LIN {X 0,Y 525.54,Z 454.136,A -85,B 0,C 180,E1 -4756.393,E2 -4756.393} C_VEL
LIN {X 0,Y 525.32,Z 467.457,A -85,B 0,C 180,E1 -4756.732,E2 -4756.732} C_VEL
LIN {X 0,Y 525.04,Z 480.774,A -85,B 0,C 180,E1 -4757.241,E2 -4757.241} C_VEL
LIN {X 0,Y 524.811,Z 492.28,A -85,B 0,C 180,E1 -4757.845,E2 -4757.845} C_VEL
LIN {X 0,Y 524.533,Z 503.565,A -85,B 0,C 180,E1 -4758.602,E2 -4758.602} C_VEL
LIN {X 0,Y 524.201,Z 514.02,A -85,B 0,C 180,E1 -4759.475,E2 -4759.475} C_VEL
LIN {X 0,Y 523.995,Z 522.569,A -85,B 0,C 180,E1 -4760.349,E2 -4760.349} C_VEL
LIN {X 0,Y 523.801,Z 530.457,A -85,B 0,C 180,E1 -4761.319,E2 -4761.319} C_VEL
LIN {X 0,Y 523.605,Z 538.16,A -85,B 0,C 180,E1 -4762.481,E2 -4762.481} C_VEL
LIN {X 0,Y 523.482,Z 545.26,A -85,B 0,C 180,E1 -4763.835,E2 -4763.835} C_VEL
LIN {X 0,Y 523.383,Z 549.983,A -85,B 0,C 180,E1 -4764.993,E2 -4764.993} C_VEL
LIN {X 0,Y 523.443,Z 553.594,A -85,B 0,C 180,E1 -4766.151,E2 -4766.151} C_VEL
LIN {X 0,Y 523.367,Z 555.454,A -85,B 0,C 180,E1 -4766.922,E2 -4766.922} C_VEL
LIN {X 0,Y 523.334,Z 556.849,A -85,B 0,C 180,E1 -4767.692,E2 -4767.692} C_VEL
LIN {X 0,Y 523.25,Z 558.451,A -85,B 0,C 180,E1 -4769.231,E2 -4769.231} C_VEL
LIN {X 0,Y 523.247,Z 558.668,A -85,B 0,C 180,E1 -4770.001,E2 -4770.001} C_VEL
LIN {X 0,Y 523.274,Z 557.846,A -85,B 0,C 180,E1 -4771.54,E2 -4771.54} C_VEL
LIN {X 0,Y 523.334,Z 556.853,A -85,B 0,C 180,E1 -4772.31,E2 -4772.31} C_VEL
LIN {X 0,Y 523.368,Z 555.459,A -85,B 0,C 180,E1 -4773.08,E2 -4773.08} C_VEL
LIN {X 0,Y 523.424,Z 552.526,A -85,B 0,C 180,E1 -4774.236,E2 -4774.236} C_VEL
LIN {X 0,Y 523.462,Z 548.553,A -85,B 0,C 180,E1 -4775.393,E2 -4775.393} C_VEL
LIN {X 0,Y 523.513,Z 542.461,A -85,B 0,C 180,E1 -4776.743,E2 -4776.743} C_VEL
LIN {X 0,Y 523.667,Z 535.765,A -85,B 0,C 180,E1 -4777.907,E2 -4777.907} C_VEL
LIN {X 0,Y 523.88,Z 527.479,A -85,B 0,C 180,E1 -4779.07,E2 -4779.07} C_VEL
LIN {X 0,Y 524.073,Z 518.984,A -85,B 0,C 180,E1 -4780.041,E2 -4780.041} C_VEL
LIN {X 0,Y 524.352,Z 508.487,A -85,B 0,C 180,E1 -4781.012,E2 -4781.012} C_VEL
LIN {X 0,Y 524.635,Z 498.224,A -85,B 0,C 180,E1 -4781.78,E2 -4781.78} C_VEL
LIN {X 0,Y 524.943,Z 486.717,A -85,B 0,C 180,E1 -4782.468,E2 -4782.468} C_VEL
LIN {X 0,Y 525.177,Z 475.022,A -85,B 0,C 180,E1 -4783.003,E2 -4783.003} C_VEL
LIN {X 0,Y 525.4,Z 461.544,A -85,B 0,C 180,E1 -4783.44,E2 -4783.44} C_VEL
LIN {X 0,Y 525.581,Z 448.167,A -85,B 0,C 180,E1 -4783.706,E2 -4783.706} C_VEL
LIN {X 0,Y 525.774,Z 355.707,A -85,B 0,C 180,E1 -4784.979,E2 -4784.979} C_VEL
LIN {X 0,Y 524.311,Z 345.996,A -85,B 0,C 180,E1 -4785.179,E2 -4785.179} C_VEL
LIN {X 0,Y 524.7,Z 326.093,A -85,B 0,C 180,E1 -4788.307,E2 -4788.307} C_VEL
LIN {X 0,Y 525.163,Z 306.772,A -85,B 0,C 180,E1 -4791.388,E2 -4791.388} C_VEL
LIN {X 0,Y 525.315,Z 297.867,A -85,B 0,C 180,E1 -4792.829,E2 -4792.829} C_VEL
LIN {X 0,Y 523.939,Z 290.22,A -85,B 0,C 180,E1 -4794.171,E2 -4794.171} C_VEL
LIN {X 0,Y 523.949,Z 290.218,A -85,B 0,C 180,E1 -4797.134,E2 -4797.134} C_VEL
LIN {X 0,Y 523.94,Z 290.224,A -85,B 0,C 180,E1 -4799.757,E2 -4799.757} C_VEL
LIN {X 0,Y 523.937,Z 290.217,A -85,B 0,C 180,E1 -4802.45,E2 -4802.45} C_VEL
LIN {X 0,Y 523.921,Z 290.217,A -85,B 0,C 180,E1 -4805.227,E2 -4805.227} C_VEL
LIN {X 0,Y 523.917,Z 290.228,A -85,B 0,C 180,E1 -4808.102,E2 -4808.102} C_VEL
LIN {X 0,Y 523.943,Z 290.214,A -85,B 0,C 180,E1 -4811.308,E2 -4811.308} C_VEL
LIN {X 0,Y 523.942,Z 290.219,A -85,B 0,C 180,E1 -4814.689,E2 -4814.689} C_VEL
LIN {X 0,Y 523.947,Z 290.215,A -85,B 0,C 180,E1 -4817.88,E2 -4817.88} C_VEL
LIN {X 0,Y 523.922,Z 290.222,A -85,B 0,C 180,E1 -4820.915,E2 -4820.915} C_VEL
LIN {X 0,Y 523.899,Z 290.22,A -85,B 0,C 180,E1 -4823.825,E2 -4823.825} C_VEL
LIN {X 0,Y 523.945,Z 290.221,A -85,B 0,C 180,E1 -4826.636,E2 -4826.636} C_VEL
LIN {X 0,Y 523.952,Z 290.216,A -85,B 0,C 180,E1 -4829.355,E2 -4829.355} C_VEL
LIN {X 0,Y 523.95,Z 290.214,A -85,B 0,C 180,E1 -4832.288,E2 -4832.288} C_VEL
LIN {X 0,Y 523.906,Z 290.224,A -85,B 0,C 180,E1 -4835.427,E2 -4835.427} C_VEL
LIN {X 0,Y 523.941,Z 290.215,A -85,B 0,C 180,E1 -4837.939,E2 -4837.939} C_VEL
LIN {X 0,Y 523.977,Z 290.21,A -85,B 0,C 180,E1 -4840.408,E2 -4840.408} C_VEL
LIN {X 0,Y 523.958,Z 290.214,A -85,B 0,C 180,E1 -4842.837,E2 -4842.837} C_VEL
LIN {X 0,Y 523.98,Z 290.214,A -85,B 0,C 180,E1 -4845.236,E2 -4845.236} C_VEL
LIN {X 0,Y 524.017,Z 290.206,A -85,B 0,C 180,E1 -4848.394,E2 -4848.394} C_VEL
LIN {X 0,Y 523.964,Z 290.217,A -85,B 0,C 180,E1 -4851.515,E2 -4851.515} C_VEL
LIN {X 0,Y 524.036,Z 290.213,A -85,B 0,C 180,E1 -4853.841,E2 -4853.841} C_VEL
LIN {X 0,Y 524.035,Z 290.203,A -85,B 0,C 180,E1 -4856.925,E2 -4856.925} C_VEL
LIN {X 0,Y 524.118,Z 290.201,A -85,B 0,C 180,E1 -4860,E2 -4860} C_VEL
LIN {X 0,Y 524.04,Z 290.202,A -85,B 0,C 180,E1 -4863.075,E2 -4863.075} C_VEL
LIN {X 0,Y 524.013,Z 290.212,A -85,B 0,C 180,E1 -4866.159,E2 -4866.159} C_VEL
LIN {X 0,Y 523.989,Z 290.209,A -85,B 0,C 180,E1 -4869.262,E2 -4869.262} C_VEL
LIN {X 0,Y 524.003,Z 290.207,A -85,B 0,C 180,E1 -4871.737,E2 -4871.737} C_VEL
LIN {X 0,Y 523.997,Z 290.212,A -85,B 0,C 180,E1 -4875.052,E2 -4875.052} C_VEL
LIN {X 0,Y 523.95,Z 290.213,A -85,B 0,C 180,E1 -4877.969,E2 -4877.969} C_VEL
LIN {X 0,Y 523.975,Z 290.213,A -85,B 0,C 180,E1 -4880.41,E2 -4880.41} C_VEL
LIN {X 0,Y 523.912,Z 290.227,A -85,B 0,C 180,E1 -4882.893,E2 -4882.893} C_VEL
LIN {X 0,Y 523.931,Z 290.22,A -85,B 0,C 180,E1 -4885.42,E2 -4885.42} C_VEL
LIN {X 0,Y 523.92,Z 290.217,A -85,B 0,C 180,E1 -4888.002,E2 -4888.002} C_VEL
LIN {X 0,Y 523.941,Z 290.218,A -85,B 0,C 180,E1 -4890.853,E2 -4890.853} C_VEL
LIN {X 0,Y 523.932,Z 290.22,A -85,B 0,C 180,E1 -4893.729,E2 -4893.729} C_VEL
LIN {X 0,Y 523.901,Z 290.219,A -85,B 0,C 180,E1 -4896.4,E2 -4896.4} C_VEL
LIN {X 0,Y 523.922,Z 290.219,A -85,B 0,C 180,E1 -4899.084,E2 -4899.084} C_VEL
LIN {X 0,Y 523.942,Z 290.218,A -85,B 0,C 180,E1 -4902.12,E2 -4902.12} C_VEL
LIN {X 0,Y 523.945,Z 290.216,A -85,B 0,C 180,E1 -4905.31,E2 -4905.31} C_VEL
LIN {X 0,Y 523.902,Z 290.219,A -85,B 0,C 180,E1 -4906.901,E2 -4906.901} C_VEL
LIN {X 0,Y 523.239,Z 290.307,A -85,B 0,C 180,E1 -4907.542,E2 -4907.542} C_VEL
LIN {X 0,Y 520.398,Z 290.666,A -85,B 0,C 180,E1 -4908.584,E2 -4908.584} C_VEL
LIN {X 0,Y 517.994,Z 290.968,A -85,B 0,C 180,E1 -4909.423,E2 -4909.423} C_VEL
LIN {X 0,Y 516.958,Z 291.094,A -85,B 0,C 180,E1 -4910.071,E2 -4910.071} C_VEL
LIN {X 0,Y 516.872,Z 291.101,A -85,B 0,C 180,E1 -4910.29,E2 -4910.29} C_VEL
LIN {X 0,Y 516.854,Z 291.097,A -85,B 0,C 180,E1 -4913.346,E2 -4913.346} C_VEL
LIN {X 0,Y 516.908,Z 291.098,A -85,B 0,C 180,E1 -4916.12,E2 -4916.12} C_VEL
LIN {X 0,Y 516.893,Z 291.094,A -85,B 0,C 180,E1 -4918.935,E2 -4918.935} C_VEL
LIN {X 0,Y 516.865,Z 291.096,A -85,B 0,C 180,E1 -4921.581,E2 -4921.581} C_VEL
LIN {X 0,Y 516.881,Z 291.098,A -85,B 0,C 180,E1 -4924.208,E2 -4924.208} C_VEL
LIN {X 0,Y 516.858,Z 291.105,A -85,B 0,C 180,E1 -4926.775,E2 -4926.775} C_VEL
LIN {X 0,Y 516.939,Z 291.087,A -85,B 0,C 180,E1 -4929.732,E2 -4929.732} C_VEL
LIN {X 0,Y 516.896,Z 291.097,A -85,B 0,C 180,E1 -4932.594,E2 -4932.594} C_VEL
LIN {X 0,Y 516.941,Z 291.096,A -85,B 0,C 180,E1 -4935.029,E2 -4935.029} C_VEL
LIN {X 0,Y 516.967,Z 291.083,A -85,B 0,C 180,E1 -4938.233,E2 -4938.233} C_VEL
LIN {X 0,Y 516.952,Z 291.095,A -85,B 0,C 180,E1 -4941.399,E2 -4941.399} C_VEL
LIN {X 0,Y 516.994,Z 291.241,A -85,B 0,C 180,E1 -4943.471,E2 -4943.471} C_VEL
LIN {X 0,Y 517.644,Z 295.731,A -85,B 0,C 180,E1 -4944.35,E2 -4944.35} C_VEL
LIN {X 0,Y 517.356,Z 311.337,A -85,B 0,C 180,E1 -4947.274,E2 -4947.274} C_VEL
LIN {X 0,Y 517.208,Z 318.952,A -85,B 0,C 180,E1 -4948.685,E2 -4948.685} C_VEL
LIN {X 0,Y 519.149,Z 330.137,A -85,B 0,C 180,E1 -4948.908,E2 -4948.908} C_VEL
LIN {X 0,Y 518.644,Z 426.311,A -85,B 0,C 180,E1 -4950.266,E2 -4950.266} C_VEL
LIN {X 0,Y 518.412,Z 439.308,A -85,B 0,C 180,E1 -4950.606,E2 -4950.606} C_VEL
LIN {X 0,Y 518.173,Z 452.352,A -85,B 0,C 180,E1 -4951.116,E2 -4951.116} C_VEL
LIN {X 0,Y 517.881,Z 464.151,A -85,B 0,C 180,E1 -4951.749,E2 -4951.749} C_VEL
LIN {X 0,Y 517.553,Z 475.474,A -85,B 0,C 180,E1 -4952.529,E2 -4952.529} C_VEL
LIN {X 0,Y 517.309,Z 485.684,A -85,B 0,C 180,E1 -4953.407,E2 -4953.407} C_VEL
LIN {X 0,Y 517.029,Z 494.082,A -85,B 0,C 180,E1 -4954.287,E2 -4954.287} C_VEL
LIN {X 0,Y 516.728,Z 503.204,A -85,B 0,C 180,E1 -4955.462,E2 -4955.462} C_VEL
LIN {X 0,Y 516.566,Z 510.863,A -85,B 0,C 180,E1 -4956.695,E2 -4956.695} C_VEL
LIN {X 0,Y 516.442,Z 516.464,A -85,B 0,C 180,E1 -4957.821,E2 -4957.821} C_VEL
LIN {X 0,Y 516.333,Z 521.149,A -85,B 0,C 180,E1 -4959.005,E2 -4959.005} C_VEL
LIN {X 0,Y 516.303,Z 524.725,A -85,B 0,C 180,E1 -4960.192,E2 -4960.192} C_VEL
LIN {X 0,Y 516.263,Z 527.383,A -85,B 0,C 180,E1 -4961.435,E2 -4961.435} C_VEL
LIN {X 0,Y 516.177,Z 528.894,A -85,B 0,C 180,E1 -4962.582,E2 -4962.582} C_VEL
LIN {X 0,Y 516.175,Z 529.466,A -85,B 0,C 180,E1 -4963.382,E2 -4963.382} C_VEL
LIN {X 0,Y 516.247,Z 529.374,A -85,B 0,C 180,E1 -4964.858,E2 -4964.858} C_VEL
LIN {X 0,Y 516.159,Z 528.598,A -85,B 0,C 180,E1 -4965.801,E2 -4965.801} C_VEL
LIN {X 0,Y 516.187,Z 527.466,A -85,B 0,C 180,E1 -4966.613,E2 -4966.613} C_VEL
LIN {X 0,Y 516.267,Z 525.342,A -85,B 0,C 180,E1 -4967.652,E2 -4967.652} C_VEL
LIN {X 0,Y 516.346,Z 521.232,A -85,B 0,C 180,E1 -4969.066,E2 -4969.066} C_VEL
LIN {X 0,Y 516.45,Z 516.137,A -85,B 0,C 180,E1 -4970.344,E2 -4970.344} C_VEL
LIN {X 0,Y 516.573,Z 510.001,A -85,B 0,C 180,E1 -4971.551,E2 -4971.551} C_VEL
LIN {X 0,Y 516.82,Z 502.019,A -85,B 0,C 180,E1 -4972.802,E2 -4972.802} C_VEL
LIN {X 0,Y 517.058,Z 493.675,A -85,B 0,C 180,E1 -4973.851,E2 -4973.851} C_VEL
LIN {X 0,Y 517.304,Z 483.311,A -85,B 0,C 180,E1 -4974.907,E2 -4974.907} C_VEL
LIN {X 0,Y 517.621,Z 473.022,A -85,B 0,C 180,E1 -4975.751,E2 -4975.751} C_VEL
LIN {X 0,Y 517.986,Z 461.243,A -85,B 0,C 180,E1 -4976.513,E2 -4976.513} C_VEL
LIN {X 0,Y 518.215,Z 448.851,A -85,B 0,C 180,E1 -4977.13,E2 -4977.13} C_VEL
LIN {X 0,Y 518.466,Z 436.346,A -85,B 0,C 180,E1 -4977.58,E2 -4977.58} C_VEL
LIN {X 0,Y 518.663,Z 423.842,A -85,B 0,C 180,E1 -4977.87,E2 -4977.87} C_VEL
LIN {X 0,Y 518.99,Z 328.564,A -85,B 0,C 180,E1 -4979.209,E2 -4979.209} C_VEL
LIN {X 0,Y 517.258,Z 318.721,A -85,B 0,C 180,E1 -4979.422,E2 -4979.422} C_VEL
LIN {X 0,Y 517.456,Z 302.677,A -85,B 0,C 180,E1 -4982.31,E2 -4982.31} C_VEL
LIN {X 0,Y 517.383,Z 294.193,A -85,B 0,C 180,E1 -4983.843,E2 -4983.843} C_VEL
LIN {X 0,Y 516.905,Z 291.101,A -85,B 0,C 180,E1 -4984.445,E2 -4984.445} C_VEL
LIN {X 0,Y 516.855,Z 291.101,A -85,B 0,C 180,E1 -4987.725,E2 -4987.725} C_VEL
LIN {X 0,Y 516.857,Z 291.106,A -85,B 0,C 180,E1 -4990.743,E2 -4990.743} C_VEL
LIN {X 0,Y 516.847,Z 291.106,A -85,B 0,C 180,E1 -4992.834,E2 -4992.834} C_VEL
LIN {X 0,Y 516.888,Z 291.103,A -85,B 0,C 180,E1 -4995.006,E2 -4995.006} C_VEL
LIN {X 0,Y 516.879,Z 291.095,A -85,B 0,C 180,E1 -4998.402,E2 -4998.402} C_VEL
LIN {X 0,Y 516.868,Z 291.106,A -85,B 0,C 180,E1 -5001.283,E2 -5001.283} C_VEL
LIN {X 0,Y 516.862,Z 291.098,A -85,B 0,C 180,E1 -5004.219,E2 -5004.219} C_VEL
LIN {X 0,Y 516.872,Z 291.093,A -85,B 0,C 180,E1 -5007.052,E2 -5007.052} C_VEL
LIN {X 0,Y 516.873,Z 291.1,A -85,B 0,C 180,E1 -5009.795,E2 -5009.795} C_VEL
LIN {X 0,Y 516.866,Z 291.097,A -85,B 0,C 180,E1 -5012.464,E2 -5012.464} C_VEL
LIN {X 0,Y 516.862,Z 291.105,A -85,B 0,C 180,E1 -5015.645,E2 -5015.645} C_VEL
LIN {X 0,Y 516.875,Z 291.096,A -85,B 0,C 180,E1 -5018.462,E2 -5018.462} C_VEL
LIN {X 0,Y 516.878,Z 291.094,A -85,B 0,C 180,E1 -5020.954,E2 -5020.954} C_VEL
LIN {X 0,Y 516.824,Z 291.102,A -85,B 0,C 180,E1 -5023.407,E2 -5023.407} C_VEL
LIN {X 0,Y 516.861,Z 291.104,A -85,B 0,C 180,E1 -5025.833,E2 -5025.833} C_VEL
LIN {X 0,Y 516.915,Z 291.097,A -85,B 0,C 180,E1 -5028.233,E2 -5028.233} C_VEL
LIN {X 0,Y 516.907,Z 291.088,A -85,B 0,C 180,E1 -5031.399,E2 -5031.399} C_VEL
LIN {X 0,Y 516.964,Z 291.089,A -85,B 0,C 180,E1 -5034.539,E2 -5034.539} C_VEL
LIN {X 0,Y 517.054,Z 291.071,A -85,B 0,C 180,E1 -5037.663,E2 -5037.663} C_VEL
LIN {X 0,Y 517.078,Z 291.072,A -85,B 0,C 180,E1 -5040.779,E2 -5040.779} C_VEL
LIN {X 0,Y 516.931,Z 291.089,A -85,B 0,C 180,E1 -5043.118,E2 -5043.118} C_VEL
LIN {X 0,Y 516.97,Z 291.087,A -85,B 0,C 180,E1 -5046.244,E2 -5046.244} C_VEL
LIN {X 0,Y 516.909,Z 291.094,A -85,B 0,C 180,E1 -5048.602,E2 -5048.602} C_VEL
LIN {X 0,Y 516.943,Z 291.085,A -85,B 0,C 180,E1 -5051.807,E2 -5051.807} C_VEL
LIN {X 0,Y 516.926,Z 291.094,A -85,B 0,C 180,E1 -5055.143,E2 -5055.143} C_VEL
LIN {X 0,Y 516.903,Z 291.088,A -85,B 0,C 180,E1 -5058.223,E2 -5058.223} C_VEL
LIN {X 0,Y 516.896,Z 291.096,A -85,B 0,C 180,E1 -5060.702,E2 -5060.702} C_VEL
LIN {X 0,Y 516.876,Z 291.094,A -85,B 0,C 180,E1 -5064.074,E2 -5064.074} C_VEL
LIN {X 0,Y 516.838,Z 291.101,A -85,B 0,C 180,E1 -5066.663,E2 -5066.663} C_VEL
LIN {X 0,Y 516.899,Z 291.099,A -85,B 0,C 180,E1 -5069.523,E2 -5069.523} C_VEL
LIN {X 0,Y 516.889,Z 291.093,A -85,B 0,C 180,E1 -5072.544,E2 -5072.544} C_VEL
LIN {X 0,Y 516.857,Z 291.104,A -85,B 0,C 180,E1 -5075.33,E2 -5075.33} C_VEL
LIN {X 0,Y 516.871,Z 291.099,A -85,B 0,C 180,E1 -5077.943,E2 -5077.943} C_VEL
LIN {X 0,Y 516.859,Z 291.098,A -85,B 0,C 180,E1 -5080.744,E2 -5080.744} C_VEL
LIN {X 0,Y 516.853,Z 291.094,A -85,B 0,C 180,E1 -5082.835,E2 -5082.835} C_VEL
LIN {X 0,Y 516.89,Z 291.093,A -85,B 0,C 180,E1 -5085.008,E2 -5085.008} C_VEL
LIN {X 0,Y 516.905,Z 291.096,A -85,B 0,C 180,E1 -5088.4,E2 -5088.4} C_VEL
LIN {X 0,Y 516.875,Z 291.098,A -85,B 0,C 180,E1 -5091.285,E2 -5091.285} C_VEL
LIN {X 0,Y 516.864,Z 291.104,A -85,B 0,C 180,E1 -5094.22,E2 -5094.22} C_VEL
LIN {X 0,Y 516.892,Z 291.095,A -85,B 0,C 180,E1 -5097.054,E2 -5097.054} C_VEL
LIN {X 0,Y 516.884,Z 291.1,A -85,B 0,C 180,E1 -5099.797,E2 -5099.797} C_VEL
LIN {X 0,Y 516.92,Z 291.099,A -85,B 0,C 180,E1 -5102.468,E2 -5102.468} C_VEL
LIN {X 0,Y 516.926,Z 291.265,A -85,B 0,C 180,E1 -5105.779,E2 -5105.779} C_VEL
LIN {X 0,Y 518.335,Z 299.595,A -85,B 0,C 180,E1 -5107.221,E2 -5107.221} C_VEL
LIN {X 0,Y 517.928,Z 316.612,A -85,B 0,C 180,E1 -5109.977,E2 -5109.977} C_VEL
LIN {X 0,Y 517.489,Z 334.423,A -85,B 0,C 180,E1 -5112.82,E2 -5112.82} C_VEL
LIN {X 0,Y 517.275,Z 346.087,A -85,B 0,C 180,E1 -5114.637,E2 -5114.637} C_VEL
LIN {X 0,Y 519.095,Z 358.575,A -85,B 0,C 180,E1 -5114.867,E2 -5114.867} C_VEL
LIN {X 0,Y 518.636,Z 453.891,A -85,B 0,C 180,E1 -5116.208,E2 -5116.208} C_VEL
LIN {X 0,Y 518.422,Z 467.226,A -85,B 0,C 180,E1 -5116.552,E2 -5116.552} C_VEL
LIN {X 0,Y 518.131,Z 479.424,A -85,B 0,C 180,E1 -5117.018,E2 -5117.018} C_VEL
LIN {X 0,Y 517.867,Z 491.836,A -85,B 0,C 180,E1 -5117.665,E2 -5117.665} C_VEL
LIN {X 0,Y 517.552,Z 503.35,A -85,B 0,C 180,E1 -5118.447,E2 -5118.447} C_VEL
LIN {X 0,Y 517.203,Z 513.807,A -85,B 0,C 180,E1 -5119.331,E2 -5119.331} C_VEL
LIN {X 0,Y 516.962,Z 522.359,A -85,B 0,C 180,E1 -5120.217,E2 -5120.217} C_VEL
LIN {X 0,Y 516.729,Z 530.248,A -85,B 0,C 180,E1 -5121.199,E2 -5121.199} C_VEL
LIN {X 0,Y 516.544,Z 537.954,A -85,B 0,C 180,E1 -5122.378,E2 -5122.378} C_VEL
LIN {X 0,Y 516.418,Z 543.657,A -85,B 0,C 180,E1 -5123.449,E2 -5123.449} C_VEL
LIN {X 0,Y 516.375,Z 548.349,A -85,B 0,C 180,E1 -5124.534,E2 -5124.534} C_VEL
LIN {X 0,Y 516.312,Z 552.321,A -85,B 0,C 180,E1 -5125.707,E2 -5125.707} C_VEL
LIN {X 0,Y 516.282,Z 555.254,A -85,B 0,C 180,E1 -5126.879,E2 -5126.879} C_VEL
LIN {X 0,Y 516.26,Z 556.65,A -85,B 0,C 180,E1 -5127.66,E2 -5127.66} C_VEL
LIN {X 0,Y 516.16,Z 558.252,A -85,B 0,C 180,E1 -5129.221,E2 -5129.221} C_VEL
LIN {X 0,Y 516.155,Z 558.469,A -85,B 0,C 180,E1 -5130.001,E2 -5130.001} C_VEL
LIN {X 0,Y 516.192,Z 557.648,A -85,B 0,C 180,E1 -5131.561,E2 -5131.561} C_VEL
LIN {X 0,Y 516.26,Z 556.656,A -85,B 0,C 180,E1 -5132.341,E2 -5132.341} C_VEL
LIN {X 0,Y 516.283,Z 555.261,A -85,B 0,C 180,E1 -5133.122,E2 -5133.122} C_VEL
LIN {X 0,Y 516.312,Z 552.327,A -85,B 0,C 180,E1 -5134.294,E2 -5134.294} C_VEL
LIN {X 0,Y 516.376,Z 548.354,A -85,B 0,C 180,E1 -5135.468,E2 -5135.468} C_VEL
LIN {X 0,Y 516.422,Z 543.143,A -85,B 0,C 180,E1 -5136.664,E2 -5136.664} C_VEL
LIN {X 0,Y 516.582,Z 536.801,A -85,B 0,C 180,E1 -5137.82,E2 -5137.82} C_VEL
LIN {X 0,Y 516.786,Z 528.768,A -85,B 0,C 180,E1 -5138.998,E2 -5138.998} C_VEL
LIN {X 0,Y 517.018,Z 520.582,A -85,B 0,C 180,E1 -5139.981,E2 -5139.981} C_VEL
LIN {X 0,Y 517.326,Z 510.6,A -85,B 0,C 180,E1 -5140.965,E2 -5140.965} C_VEL
LIN {X 0,Y 517.629,Z 500.75,A -85,B 0,C 180,E1 -5141.752,E2 -5141.752} C_VEL
LIN {X 0,Y 517.917,Z 489.613,A -85,B 0,C 180,E1 -5142.465,E2 -5142.465} C_VEL
LIN {X 0,Y 518.178,Z 477.16,A -85,B 0,C 180,E1 -5143.082,E2 -5143.082} C_VEL
LIN {X 0,Y 518.439,Z 464.063,A -85,B 0,C 180,E1 -5143.549,E2 -5143.549} C_VEL
LIN {X 0,Y 518.659,Z 450.968,A -85,B 0,C 180,E1 -5143.843,E2 -5143.843} C_VEL
LIN {X 0,Y 518.991,Z 356.872,A -85,B 0,C 180,E1 -5145.16,E2 -5145.16} C_VEL
LIN {X 0,Y 517.289,Z 345.951,A -85,B 0,C 180,E1 -5145.366,E2 -5145.366} C_VEL
LIN {X 0,Y 517.746,Z 325.651,A -85,B 0,C 180,E1 -5148.603,E2 -5148.603} C_VEL
LIN {X 0,Y 518.203,Z 307.858,A -85,B 0,C 180,E1 -5151.481,E2 -5151.481} C_VEL
LIN {X 0,Y 518.355,Z 299.1,A -85,B 0,C 180,E1 -5152.915,E2 -5152.915} C_VEL
LIN {X 0,Y 516.884,Z 291.099,A -85,B 0,C 180,E1 -5154.317,E2 -5154.317} C_VEL
LIN {X 0,Y 516.926,Z 291.098,A -85,B 0,C 180,E1 -5157.533,E2 -5157.533} C_VEL
LIN {X 0,Y 516.89,Z 291.097,A -85,B 0,C 180,E1 -5160.204,E2 -5160.204} C_VEL
LIN {X 0,Y 516.899,Z 291.092,A -85,B 0,C 180,E1 -5162.947,E2 -5162.947} C_VEL
LIN {X 0,Y 516.871,Z 291.101,A -85,B 0,C 180,E1 -5165.781,E2 -5165.781} C_VEL
LIN {X 0,Y 516.881,Z 291.096,A -85,B 0,C 180,E1 -5168.716,E2 -5168.716} C_VEL
LIN {X 0,Y 516.905,Z 291.094,A -85,B 0,C 180,E1 -5171.776,E2 -5171.776} C_VEL
LIN {X 0,Y 516.899,Z 291.093,A -85,B 0,C 180,E1 -5175.007,E2 -5175.007} C_VEL
LIN {X 0,Y 516.914,Z 291.098,A -85,B 0,C 180,E1 -5178.399,E2 -5178.399} C_VEL
LIN {X 0,Y 516.882,Z 291.095,A -85,B 0,C 180,E1 -5181.284,E2 -5181.284} C_VEL
LIN {X 0,Y 516.871,Z 291.097,A -85,B 0,C 180,E1 -5184.219,E2 -5184.219} C_VEL
LIN {X 0,Y 516.899,Z 291.098,A -85,B 0,C 180,E1 -5187.053,E2 -5187.053} C_VEL
LIN {X 0,Y 516.89,Z 291.093,A -85,B 0,C 180,E1 -5189.796,E2 -5189.796} C_VEL
LIN {X 0,Y 516.903,Z 291.093,A -85,B 0,C 180,E1 -5192.466,E2 -5192.466} C_VEL
LIN {X 0,Y 516.849,Z 291.107,A -85,B 0,C 180,E1 -5195.068,E2 -5195.068} C_VEL
LIN {X 0,Y 516.873,Z 291.099,A -85,B 0,C 180,E1 -5197.621,E2 -5197.621} C_VEL
LIN {X 0,Y 516.935,Z 291.088,A -85,B 0,C 180,E1 -5200.13,E2 -5200.13} C_VEL
LIN {X 0,Y 516.909,Z 291.09,A -85,B 0,C 180,E1 -5202.595,E2 -5202.595} C_VEL
LIN {X 0,Y 516.946,Z 291.088,A -85,B 0,C 180,E1 -5205.03,E2 -5205.03} C_VEL
LIN {X 0,Y 516.97,Z 291.085,A -85,B 0,C 180,E1 -5208.234,E2 -5208.234} C_VEL
LIN {X 0,Y 516.939,Z 291.091,A -85,B 0,C 180,E1 -5211.399,E2 -5211.399} C_VEL
LIN {X 0,Y 517.002,Z 291.087,A -85,B 0,C 180,E1 -5213.757,E2 -5213.757} C_VEL
LIN {X 0,Y 517.084,Z 291.073,A -85,B 0,C 180,E1 -5217.663,E2 -5217.663} C_VEL
LIN {X 0,Y 517.091,Z 291.069,A -85,B 0,C 180,E1 -5220.779,E2 -5220.779} C_VEL
LIN {X 0,Y 516.983,Z 291.081,A -85,B 0,C 180,E1 -5223.117,E2 -5223.117} C_VEL
LIN {X 0,Y 516.978,Z 291.09,A -85,B 0,C 180,E1 -5226.243,E2 -5226.243} C_VEL
LIN {X 0,Y 516.944,Z 291.086,A -85,B 0,C 180,E1 -5229.389,E2 -5229.389} C_VEL
LIN {X 0,Y 516.955,Z 291.085,A -85,B 0,C 180,E1 -5231.807,E2 -5231.807} C_VEL
LIN {X 0,Y 516.95,Z 291.088,A -85,B 0,C 180,E1 -5235.147,E2 -5235.147} C_VEL
LIN {X 0,Y 516.918,Z 291.091,A -85,B 0,C 180,E1 -5238.222,E2 -5238.222} C_VEL
LIN {X 0,Y 516.915,Z 291.096,A -85,B 0,C 180,E1 -5240.701,E2 -5240.701} C_VEL
LIN {X 0,Y 516.891,Z 291.092,A -85,B 0,C 180,E1 -5244.073,E2 -5244.073} C_VEL
LIN {X 0,Y 516.9,Z 291.094,A -85,B 0,C 180,E1 -5246.659,E2 -5246.659} C_VEL
LIN {X 0,Y 516.911,Z 291.096,A -85,B 0,C 180,E1 -5249.523,E2 -5249.523} C_VEL
LIN {X 0,Y 516.896,Z 291.092,A -85,B 0,C 180,E1 -5252.543,E2 -5252.543} C_VEL
LIN {X 0,Y 516.866,Z 291.104,A -85,B 0,C 180,E1 -5255.329,E2 -5255.329} C_VEL
LIN {X 0,Y 516.881,Z 291.098,A -85,B 0,C 180,E1 -5257.942,E2 -5257.942} C_VEL
LIN {X 0,Y 516.882,Z 291.094,A -85,B 0,C 180,E1 -5260.742,E2 -5260.742} C_VEL
LIN {X 0,Y 516.883,Z 291.102,A -85,B 0,C 180,E1 -5263.903,E2 -5263.903} C_VEL
LIN {X 0,Y 516.85,Z 291.098,A -85,B 0,C 180,E1 -5266.902,E2 -5266.902} C_VEL
LIN {X 0,Y 516.886,Z 291.097,A -85,B 0,C 180,E1 -5269.589,E2 -5269.589} C_VEL
LIN {X 0,Y 516.872,Z 291.101,A -85,B 0,C 180,E1 -5270.29,E2 -5270.29} C_VEL
LIN {X 0,Y 516.201,Z 291.181,A -85,B 0,C 180,E1 -5270.94,E2 -5270.94} C_VEL
LIN {X 0,Y 513.347,Z 291.542,A -85,B 0,C 180,E1 -5271.996,E2 -5271.996} C_VEL
LIN {X 0,Y 510.934,Z 291.841,A -85,B 0,C 180,E1 -5272.846,E2 -5272.846} C_VEL
LIN {X 0,Y 509.894,Z 291.967,A -85,B 0,C 180,E1 -5273.503,E2 -5273.503} C_VEL
LIN {X 0,Y 509.807,Z 291.977,A -85,B 0,C 180,E1 -5273.725,E2 -5273.725} C_VEL
LIN {X 0,Y 509.86,Z 291.974,A -85,B 0,C 180,E1 -5276.539,E2 -5276.539} C_VEL
LIN {X 0,Y 509.847,Z 291.97,A -85,B 0,C 180,E1 -5279.334,E2 -5279.334} C_VEL
LIN {X 0,Y 509.852,Z 291.973,A -85,B 0,C 180,E1 -5282.051,E2 -5282.051} C_VEL
LIN {X 0,Y 509.809,Z 291.983,A -85,B 0,C 180,E1 -5284.7,E2 -5284.7} C_VEL
LIN {X 0,Y 509.826,Z 291.973,A -85,B 0,C 180,E1 -5287.458,E2 -5287.458} C_VEL
LIN {X 0,Y 509.916,Z 291.961,A -85,B 0,C 180,E1 -5289.844,E2 -5289.844} C_VEL
LIN {X 0,Y 509.865,Z 291.974,A -85,B 0,C 180,E1 -5293.173,E2 -5293.173} C_VEL
LIN {X 0,Y 509.857,Z 291.97,A -85,B 0,C 180,E1 -5295.633,E2 -5295.633} C_VEL
LIN {X 0,Y 509.909,Z 291.968,A -85,B 0,C 180,E1 -5298.874,E2 -5298.874} C_VEL
LIN {X 0,Y 509.92,Z 291.966,A -85,B 0,C 180,E1 -5302.077,E2 -5302.077} C_VEL
LIN {X 0,Y 509.958,Z 292.135,A -85,B 0,C 180,E1 -5303.343,E2 -5303.343} C_VEL
LIN {X 0,Y 510.664,Z 296.834,A -85,B 0,C 180,E1 -5304.273,E2 -5304.273} C_VEL
LIN {X 0,Y 510.379,Z 311.463,A -85,B 0,C 180,E1 -5307.039,E2 -5307.039} C_VEL
LIN {X 0,Y 510.242,Z 319.101,A -85,B 0,C 180,E1 -5308.47,E2 -5308.47} C_VEL
LIN {X 0,Y 512.269,Z 330.125,A -85,B 0,C 180,E1 -5308.697,E2 -5308.697} C_VEL
LIN {X 0,Y 511.753,Z 426.291,A -85,B 0,C 180,E1 -5310.073,E2 -5310.073} C_VEL
LIN {X 0,Y 511.534,Z 439.338,A -85,B 0,C 180,E1 -5310.417,E2 -5310.417} C_VEL
LIN {X 0,Y 511.263,Z 452.439,A -85,B 0,C 180,E1 -5310.935,E2 -5310.935} C_VEL
LIN {X 0,Y 510.938,Z 464.274,A -85,B 0,C 180,E1 -5311.576,E2 -5311.576} C_VEL
LIN {X 0,Y 510.584,Z 475.614,A -85,B 0,C 180,E1 -5312.366,E2 -5312.366} C_VEL
LIN {X 0,Y 510.319,Z 485.833,A -85,B 0,C 180,E1 -5313.256,E2 -5313.256} C_VEL
LIN {X 0,Y 510.003,Z 494.244,A -85,B 0,C 180,E1 -5314.148,E2 -5314.148} C_VEL
LIN {X 0,Y 509.749,Z 502.011,A -85,B 0,C 180,E1 -5315.141,E2 -5315.141} C_VEL
LIN {X 0,Y 509.577,Z 509.605,A -85,B 0,C 180,E1 -5316.334,E2 -5316.334} C_VEL
LIN {X 0,Y 509.41,Z 515.734,A -85,B 0,C 180,E1 -5317.53,E2 -5317.53} C_VEL
LIN {X 0,Y 509.278,Z 520.613,A -85,B 0,C 180,E1 -5318.73,E2 -5318.73} C_VEL
LIN {X 0,Y 509.23,Z 524.372,A -85,B 0,C 180,E1 -5319.933,E2 -5319.933} C_VEL
LIN {X 0,Y 509.174,Z 527.725,A -85,B 0,C 180,E1 -5321.48,E2 -5321.48} C_VEL
LIN {X 0,Y 509.099,Z 529.286,A -85,B 0,C 180,E1 -5322.76,E2 -5322.76} C_VEL
LIN {X 0,Y 509.085,Z 529.718,A -85,B 0,C 180,E1 -5323.572,E2 -5323.572} C_VEL
LIN {X 0,Y 509.148,Z 529.536,A -85,B 0,C 180,E1 -5324.93,E2 -5324.93} C_VEL
LIN {X 0,Y 509.063,Z 528.566,A -85,B 0,C 180,E1 -5326.028,E2 -5326.028} C_VEL
LIN {X 0,Y 509.105,Z 527.296,A -85,B 0,C 180,E1 -5326.851,E2 -5326.851} C_VEL
LIN {X 0,Y 509.197,Z 525.411,A -85,B 0,C 180,E1 -5327.76,E2 -5327.76} C_VEL
LIN {X 0,Y 509.264,Z 522.13,A -85,B 0,C 180,E1 -5328.923,E2 -5328.923} C_VEL
LIN {X 0,Y 509.393,Z 517.147,A -85,B 0,C 180,E1 -5330.252,E2 -5330.252} C_VEL
LIN {X 0,Y 509.484,Z 511.396,A -85,B 0,C 180,E1 -5331.44,E2 -5331.44} C_VEL
LIN {X 0,Y 509.738,Z 503.68,A -85,B 0,C 180,E1 -5332.708,E2 -5332.708} C_VEL
LIN {X 0,Y 509.978,Z 495.696,A -85,B 0,C 180,E1 -5333.771,E2 -5333.771} C_VEL
LIN {X 0,Y 510.298,Z 486.306,A -85,B 0,C 180,E1 -5334.793,E2 -5334.793} C_VEL
LIN {X 0,Y 510.617,Z 476.044,A -85,B 0,C 180,E1 -5335.693,E2 -5335.693} C_VEL
LIN {X 0,Y 510.936,Z 465.895,A -85,B 0,C 180,E1 -5336.413,E2 -5336.413} C_VEL
LIN {X 0,Y 511.232,Z 453.865,A -85,B 0,C 180,E1 -5337.088,E2 -5337.088} C_VEL
LIN {X 0,Y 511.447,Z 442.37,A -85,B 0,C 180,E1 -5337.574,E2 -5337.574} C_VEL
LIN {X 0,Y 511.682,Z 429.048,A -85,B 0,C 180,E1 -5337.959,E2 -5337.959} C_VEL
LIN {X 0,Y 511.847,Z 410.339,A -85,B 0,C 180,E1 -5338.262,E2 -5338.262} C_VEL
LIN {X 0,Y 512.232,Z 329.911,A -85,B 0,C 180,E1 -5339.398,E2 -5339.398} C_VEL
LIN {X 0,Y 510.249,Z 318.946,A -85,B 0,C 180,E1 -5339.624,E2 -5339.624} C_VEL
LIN {X 0,Y 510.471,Z 302.1,A -85,B 0,C 180,E1 -5342.68,E2 -5342.68} C_VEL
LIN {X 0,Y 510.413,Z 295.471,A -85,B 0,C 180,E1 -5343.893,E2 -5343.893} C_VEL
LIN {X 0,Y 509.861,Z 291.978,A -85,B 0,C 180,E1 -5344.591,E2 -5344.591} C_VEL
LIN {X 0,Y 509.81,Z 291.981,A -85,B 0,C 180,E1 -5347.34,E2 -5347.34} C_VEL
LIN {X 0,Y 509.811,Z 291.979,A -85,B 0,C 180,E1 -5350.384,E2 -5350.384} C_VEL
LIN {X 0,Y 509.794,Z 291.987,A -85,B 0,C 180,E1 -5353.059,E2 -5353.059} C_VEL
LIN {X 0,Y 509.814,Z 291.977,A -85,B 0,C 180,E1 -5355.793,E2 -5355.793} C_VEL
LIN {X 0,Y 509.823,Z 291.975,A -85,B 0,C 180,E1 -5358.571,E2 -5358.571} C_VEL
LIN {X 0,Y 509.841,Z 291.974,A -85,B 0,C 180,E1 -5361.786,E2 -5361.786} C_VEL
LIN {X 0,Y 509.82,Z 291.975,A -85,B 0,C 180,E1 -5364.621,E2 -5364.621} C_VEL
LIN {X 0,Y 509.851,Z 291.975,A -85,B 0,C 180,E1 -5367.48,E2 -5367.48} C_VEL
LIN {X 0,Y 509.849,Z 291.97,A -85,B 0,C 180,E1 -5370.274,E2 -5370.274} C_VEL
LIN {X 0,Y 509.811,Z 291.977,A -85,B 0,C 180,E1 -5372.94,E2 -5372.94} C_VEL
LIN {X 0,Y 509.824,Z 291.98,A -85,B 0,C 180,E1 -5375.572,E2 -5375.572} C_VEL
LIN {X 0,Y 509.812,Z 291.978,A -85,B 0,C 180,E1 -5378.148,E2 -5378.148} C_VEL
LIN {X 0,Y 509.844,Z 291.971,A -85,B 0,C 180,E1 -5380.681,E2 -5380.681} C_VEL
LIN {X 0,Y 509.778,Z 291.978,A -85,B 0,C 180,E1 -5383.171,E2 -5383.171} C_VEL
LIN {X 0,Y 509.834,Z 291.976,A -85,B 0,C 180,E1 -5385.633,E2 -5385.633} C_VEL
LIN {X 0,Y 509.879,Z 291.975,A -85,B 0,C 180,E1 -5388.131,E2 -5388.131} C_VEL
LIN {X 0,Y 509.861,Z 291.965,A -85,B 0,C 180,E1 -5391.279,E2 -5391.279} C_VEL
LIN {X 0,Y 509.884,Z 291.967,A -85,B 0,C 180,E1 -5393.669,E2 -5393.669} C_VEL
LIN {X 0,Y 509.873,Z 291.967,A -85,B 0,C 180,E1 -5396.84,E2 -5396.84} C_VEL
LIN {X 0,Y 509.916,Z 291.97,A -85,B 0,C 180,E1 -5398.421,E2 -5398.421} C_VEL
LIN {X 0,Y 510.027,Z 291.95,A -85,B 0,C 180,E1 -5400.79,E2 -5400.79} C_VEL
LIN {X 0,Y 509.875,Z 291.967,A -85,B 0,C 180,E1 -5403.161,E2 -5403.161} C_VEL
LIN {X 0,Y 509.924,Z 291.966,A -85,B 0,C 180,E1 -5406.33,E2 -5406.33} C_VEL
LIN {X 0,Y 509.842,Z 291.971,A -85,B 0,C 180,E1 -5409.522,E2 -5409.522} C_VEL
LIN {X 0,Y 509.895,Z 291.963,A -85,B 0,C 180,E1 -5411.932,E2 -5411.932} C_VEL
LIN {X 0,Y 509.886,Z 291.969,A -85,B 0,C 180,E1 -5415.242,E2 -5415.242} C_VEL
LIN {X 0,Y 509.847,Z 291.968,A -85,B 0,C 180,E1 -5418.484,E2 -5418.484} C_VEL
LIN {X 0,Y 509.837,Z 291.98,A -85,B 0,C 180,E1 -5421.002,E2 -5421.002} C_VEL
LIN {X 0,Y 509.81,Z 291.978,A -85,B 0,C 180,E1 -5423.565,E2 -5423.565} C_VEL
LIN {X 0,Y 509.811,Z 291.975,A -85,B 0,C 180,E1 -5426.358,E2 -5426.358} C_VEL
LIN {X 0,Y 509.842,Z 291.973,A -85,B 0,C 180,E1 -5428.847,E2 -5428.847} C_VEL
LIN {X 0,Y 509.811,Z 291.981,A -85,B 0,C 180,E1 -5431.591,E2 -5431.591} C_VEL
LIN {X 0,Y 509.84,Z 291.972,A -85,B 0,C 180,E1 -5434.415,E2 -5434.415} C_VEL
LIN {X 0,Y 509.801,Z 291.983,A -85,B 0,C 180,E1 -5437.342,E2 -5437.342} C_VEL
LIN {X 0,Y 509.812,Z 291.977,A -85,B 0,C 180,E1 -5440.385,E2 -5440.385} C_VEL
LIN {X 0,Y 509.799,Z 291.974,A -85,B 0,C 180,E1 -5443.061,E2 -5443.061} C_VEL
LIN {X 0,Y 509.818,Z 291.984,A -85,B 0,C 180,E1 -5445.794,E2 -5445.794} C_VEL
LIN {X 0,Y 509.848,Z 291.974,A -85,B 0,C 180,E1 -5448.575,E2 -5448.575} C_VEL
LIN {X 0,Y 509.846,Z 291.979,A -85,B 0,C 180,E1 -5451.788,E2 -5451.788} C_VEL
LIN {X 0,Y 509.824,Z 291.975,A -85,B 0,C 180,E1 -5454.623,E2 -5454.623} C_VEL
LIN {X 0,Y 509.859,Z 291.972,A -85,B 0,C 180,E1 -5457.482,E2 -5457.482} C_VEL
LIN {X 0,Y 509.856,Z 291.977,A -85,B 0,C 180,E1 -5460.275,E2 -5460.275} C_VEL
LIN {X 0,Y 509.872,Z 291.974,A -85,B 0,C 180,E1 -5462.945,E2 -5462.945} C_VEL
LIN {X 0,Y 509.853,Z 292.012,A -85,B 0,C 180,E1 -5465.574,E2 -5465.574} C_VEL
LIN {X 0,Y 511.359,Z 300.354,A -85,B 0,C 180,E1 -5467.049,E2 -5467.049} C_VEL
LIN {X 0,Y 511.014,Z 315.639,A -85,B 0,C 180,E1 -5469.569,E2 -5469.569} C_VEL
LIN {X 0,Y 510.503,Z 334.207,A -85,B 0,C 180,E1 -5472.578,E2 -5472.578} C_VEL
LIN {X 0,Y 510.239,Z 345.662,A -85,B 0,C 180,E1 -5474.416,E2 -5474.416} C_VEL
LIN {X 0,Y 512.255,Z 359.615,A -85,B 0,C 180,E1 -5474.678,E2 -5474.678} C_VEL
LIN {X 0,Y 511.761,Z 453.644,A -85,B 0,C 180,E1 -5476.019,E2 -5476.019} C_VEL
LIN {X 0,Y 511.523,Z 466.993,A -85,B 0,C 180,E1 -5476.367,E2 -5476.367} C_VEL
LIN {X 0,Y 511.174,Z 480.325,A -85,B 0,C 180,E1 -5476.889,E2 -5476.889} C_VEL
LIN {X 0,Y 510.903,Z 491.791,A -85,B 0,C 180,E1 -5477.506,E2 -5477.506} C_VEL
LIN {X 0,Y 510.57,Z 503.134,A -85,B 0,C 180,E1 -5478.286,E2 -5478.286} C_VEL
LIN {X 0,Y 510.212,Z 513.595,A -85,B 0,C 180,E1 -5479.183,E2 -5479.183} C_VEL
LIN {X 0,Y 509.94,Z 522.148,A -85,B 0,C 180,E1 -5480.081,E2 -5480.081} C_VEL
LIN {X 0,Y 509.681,Z 530.04,A -85,B 0,C 180,E1 -5481.077,E2 -5481.077} C_VEL
LIN {X 0,Y 509.479,Z 537.748,A -85,B 0,C 180,E1 -5482.271,E2 -5482.271} C_VEL
LIN {X 0,Y 509.318,Z 543.986,A -85,B 0,C 180,E1 -5483.474,E2 -5483.474} C_VEL
LIN {X 0,Y 509.243,Z 549.579,A -85,B 0,C 180,E1 -5484.854,E2 -5484.854} C_VEL
LIN {X 0,Y 509.245,Z 553.191,A -85,B 0,C 180,E1 -5486.044,E2 -5486.044} C_VEL
LIN {X 0,Y 509.2,Z 555.054,A -85,B 0,C 180,E1 -5486.836,E2 -5486.836} C_VEL
LIN {X 0,Y 509.189,Z 556.45,A -85,B 0,C 180,E1 -5487.628,E2 -5487.628} C_VEL
LIN {X 0,Y 509.073,Z 558.054,A -85,B 0,C 180,E1 -5489.21,E2 -5489.21} C_VEL
LIN {X 0,Y 509.066,Z 558.271,A -85,B 0,C 180,E1 -5490.001,E2 -5490.001} C_VEL
LIN {X 0,Y 509.112,Z 557.45,A -85,B 0,C 180,E1 -5491.583,E2 -5491.583} C_VEL
LIN {X 0,Y 509.189,Z 556.458,A -85,B 0,C 180,E1 -5492.374,E2 -5492.374} C_VEL
LIN {X 0,Y 509.201,Z 555.063,A -85,B 0,C 180,E1 -5493.165,E2 -5493.165} C_VEL
LIN {X 0,Y 509.204,Z 552.128,A -85,B 0,C 180,E1 -5494.354,E2 -5494.354} C_VEL
LIN {X 0,Y 509.293,Z 548.155,A -85,B 0,C 180,E1 -5495.544,E2 -5495.544} C_VEL
LIN {X 0,Y 509.397,Z 542.144,A -85,B 0,C 180,E1 -5496.914,E2 -5496.914} C_VEL
LIN {X 0,Y 509.545,Z 535.362,A -85,B 0,C 180,E1 -5498.128,E2 -5498.128} C_VEL
LIN {X 0,Y 509.783,Z 527.074,A -85,B 0,C 180,E1 -5499.323,E2 -5499.323} C_VEL
LIN {X 0,Y 510.016,Z 518.575,A -85,B 0,C 180,E1 -5500.32,E2 -5500.32} C_VEL
LIN {X 0,Y 510.395,Z 508.075,A -85,B 0,C 180,E1 -5501.317,E2 -5501.317} C_VEL
LIN {X 0,Y 510.688,Z 497.802,A -85,B 0,C 180,E1 -5502.107,E2 -5502.107} C_VEL
LIN {X 0,Y 511.05,Z 486.294,A -85,B 0,C 180,E1 -5502.813,E2 -5502.813} C_VEL
LIN {X 0,Y 511.359,Z 474.585,A -85,B 0,C 180,E1 -5503.361,E2 -5503.361} C_VEL
LIN {X 0,Y 511.592,Z 461.09,A -85,B 0,C 180,E1 -5503.81,E2 -5503.81} C_VEL
LIN {X 0,Y 511.819,Z 447.66,A -85,B 0,C 180,E1 -5504.082,E2 -5504.082} C_VEL
LIN {X 0,Y 512.17,Z 357.903,A -85,B 0,C 180,E1 -5505.35,E2 -5505.35} C_VEL
LIN {X 0,Y 510.259,Z 345.664,A -85,B 0,C 180,E1 -5505.597,E2 -5505.597} C_VEL
LIN {X 0,Y 510.755,Z 326.736,A -85,B 0,C 180,E1 -5508.659,E2 -5508.659} C_VEL
LIN {X 0,Y 511.252,Z 308.917,A -85,B 0,C 180,E1 -5511.576,E2 -5511.576} C_VEL
LIN {X 0,Y 511.433,Z 300.494,A -85,B 0,C 180,E1 -5512.971,E2 -5512.971} C_VEL
LIN {X 0,Y 509.856,Z 291.975,A -85,B 0,C 180,E1 -5514.473,E2 -5514.473} C_VEL
LIN {X 0,Y 509.878,Z 291.971,A -85,B 0,C 180,E1 -5517.057,E2 -5517.057} C_VEL
LIN {X 0,Y 509.861,Z 291.978,A -85,B 0,C 180,E1 -5519.751,E2 -5519.751} C_VEL
LIN {X 0,Y 509.877,Z 291.966,A -85,B 0,C 180,E1 -5522.774,E2 -5522.774} C_VEL
LIN {X 0,Y 509.826,Z 291.976,A -85,B 0,C 180,E1 -5525.578,E2 -5525.578} C_VEL
LIN {X 0,Y 509.852,Z 291.976,A -85,B 0,C 180,E1 -5528.338,E2 -5528.338} C_VEL
LIN {X 0,Y 509.848,Z 291.97,A -85,B 0,C 180,E1 -5531.427,E2 -5531.427} C_VEL
LIN {X 0,Y 509.843,Z 291.976,A -85,B 0,C 180,E1 -5534.67,E2 -5534.67} C_VEL
LIN {X 0,Y 509.854,Z 291.973,A -85,B 0,C 180,E1 -5538.104,E2 -5538.104} C_VEL
LIN {X 0,Y 509.849,Z 291.979,A -85,B 0,C 180,E1 -5540.647,E2 -5540.647} C_VEL
LIN {X 0,Y 509.813,Z 291.974,A -85,B 0,C 180,E1 -5543.646,E2 -5543.646} C_VEL
LIN {X 0,Y 509.862,Z 291.973,A -85,B 0,C 180,E1 -5546.539,E2 -5546.539} C_VEL
LIN {X 0,Y 509.846,Z 291.974,A -85,B 0,C 180,E1 -5549.334,E2 -5549.334} C_VEL
LIN {X 0,Y 509.854,Z 291.969,A -85,B 0,C 180,E1 -5552.052,E2 -5552.052} C_VEL
LIN {X 0,Y 509.807,Z 291.978,A -85,B 0,C 180,E1 -5554.7,E2 -5554.7} C_VEL
LIN {X 0,Y 509.829,Z 291.979,A -85,B 0,C 180,E1 -5557.458,E2 -5557.458} C_VEL
LIN {X 0,Y 509.92,Z 291.963,A -85,B 0,C 180,E1 -5559.845,E2 -5559.845} C_VEL
LIN {X 0,Y 509.876,Z 291.972,A -85,B 0,C 180,E1 -5563.174,E2 -5563.174} C_VEL
LIN {X 0,Y 509.864,Z 291.977,A -85,B 0,C 180,E1 -5565.634,E2 -5565.634} C_VEL
LIN {X 0,Y 509.915,Z 291.962,A -85,B 0,C 180,E1 -5568.874,E2 -5568.874} C_VEL
LIN {X 0,Y 509.918,Z 291.967,A -85,B 0,C 180,E1 -5572.078,E2 -5572.078} C_VEL
LIN {X 0,Y 509.977,Z 291.956,A -85,B 0,C 180,E1 -5574.464,E2 -5574.464} C_VEL
LIN {X 0,Y 510.053,Z 291.948,A -85,B 0,C 180,E1 -5577.631,E2 -5577.631} C_VEL
LIN {X 0,Y 510.06,Z 291.952,A -85,B 0,C 180,E1 -5580,E2 -5580} C_VEL
LIN {X 0,Y 510.052,Z 291.952,A -85,B 0,C 180,E1 -5582.369,E2 -5582.369} C_VEL
LIN {X 0,Y 509.966,Z 291.956,A -85,B 0,C 180,E1 -5585.536,E2 -5585.536} C_VEL
LIN {X 0,Y 509.912,Z 291.967,A -85,B 0,C 180,E1 -5588.72,E2 -5588.72} C_VEL
LIN {X 0,Y 509.908,Z 291.964,A -85,B 0,C 180,E1 -5591.931,E2 -5591.931} C_VEL
LIN {X 0,Y 509.897,Z 291.966,A -85,B 0,C 180,E1 -5595.242,E2 -5595.242} C_VEL
LIN {X 0,Y 509.863,Z 291.973,A -85,B 0,C 180,E1 -5598.483,E2 -5598.483} C_VEL
LIN {X 0,Y 509.853,Z 291.978,A -85,B 0,C 180,E1 -5601.001,E2 -5601.001} C_VEL
LIN {X 0,Y 509.823,Z 291.975,A -85,B 0,C 180,E1 -5603.564,E2 -5603.564} C_VEL
LIN {X 0,Y 509.882,Z 291.966,A -85,B 0,C 180,E1 -5606.371,E2 -5606.371} C_VEL
LIN {X 0,Y 509.86,Z 291.971,A -85,B 0,C 180,E1 -5609.726,E2 -5609.726} C_VEL
LIN {X 0,Y 509.869,Z 291.969,A -85,B 0,C 180,E1 -5612.773,E2 -5612.773} C_VEL
LIN {X 0,Y 509.825,Z 291.981,A -85,B 0,C 180,E1 -5615.578,E2 -5615.578} C_VEL
LIN {X 0,Y 509.851,Z 291.97,A -85,B 0,C 180,E1 -5618.338,E2 -5618.338} C_VEL
LIN {X 0,Y 509.853,Z 291.975,A -85,B 0,C 180,E1 -5621.426,E2 -5621.426} C_VEL
LIN {X 0,Y 509.841,Z 291.971,A -85,B 0,C 180,E1 -5624.67,E2 -5624.67} C_VEL
LIN {X 0,Y 509.852,Z 291.977,A -85,B 0,C 180,E1 -5628.104,E2 -5628.104} C_VEL
LIN {X 0,Y 509.839,Z 291.973,A -85,B 0,C 180,E1 -5630.646,E2 -5630.646} C_VEL
LIN {X 0,Y 509.807,Z 291.977,A -85,B 0,C 180,E1 -5633.725,E2 -5633.725} C_VEL
LIN {X 0,Y 509.148,Z 292.064,A -85,B 0,C 180,E1 -5634.385,E2 -5634.385} C_VEL
LIN {X 0,Y 506.343,Z 292.409,A -85,B 0,C 180,E1 -5635.457,E2 -5635.457} C_VEL
LIN {X 0,Y 503.957,Z 292.713,A -85,B 0,C 180,E1 -5636.321,E2 -5636.321} C_VEL
LIN {X 0,Y 502.909,Z 292.836,A -85,B 0,C 180,E1 -5636.987,E2 -5636.987} C_VEL
LIN {X 0,Y 502.811,Z 292.847,A -85,B 0,C 180,E1 -5637.213,E2 -5637.213} C_VEL
LIN {X 0,Y 502.817,Z 292.85,A -85,B 0,C 180,E1 -5640.065,E2 -5640.065} C_VEL
LIN {X 0,Y 502.845,Z 292.842,A -85,B 0,C 180,E1 -5643.443,E2 -5643.443} C_VEL
LIN {X 0,Y 502.788,Z 292.855,A -85,B 0,C 180,E1 -5646.959,E2 -5646.959} C_VEL
LIN {X 0,Y 502.835,Z 292.844,A -85,B 0,C 180,E1 -5649.548,E2 -5649.548} C_VEL
LIN {X 0,Y 502.818,Z 292.846,A -85,B 0,C 180,E1 -5652.091,E2 -5652.091} C_VEL
LIN {X 0,Y 502.841,Z 292.846,A -85,B 0,C 180,E1 -5655.428,E2 -5655.428} C_VEL
LIN {X 0,Y 502.874,Z 292.842,A -85,B 0,C 180,E1 -5658.716,E2 -5658.716} C_VEL
LIN {X 0,Y 502.88,Z 292.844,A -85,B 0,C 180,E1 -5661.966,E2 -5661.966} C_VEL
LIN {X 0,Y 502.93,Z 292.958,A -85,B 0,C 180,E1 -5663.198,E2 -5663.198} C_VEL
LIN {X 0,Y 503.68,Z 297.948,A -85,B 0,C 180,E1 -5664.193,E2 -5664.193} C_VEL
LIN {X 0,Y 503.385,Z 312.635,A -85,B 0,C 180,E1 -5666.998,E2 -5666.998} C_VEL
LIN {X 0,Y 503.271,Z 319.247,A -85,B 0,C 180,E1 -5668.249,E2 -5668.249} C_VEL
LIN {X 0,Y 505.463,Z 331.693,A -85,B 0,C 180,E1 -5668.505,E2 -5668.505} C_VEL
LIN {X 0,Y 504.893,Z 426.241,A -85,B 0,C 180,E1 -5669.875,E2 -5669.875} C_VEL
LIN {X 0,Y 504.647,Z 439.381,A -85,B 0,C 180,E1 -5670.224,E2 -5670.224} C_VEL
LIN {X 0,Y 504.378,Z 452.512,A -85,B 0,C 180,E1 -5670.748,E2 -5670.748} C_VEL
LIN {X 0,Y 504.015,Z 464.391,A -85,B 0,C 180,E1 -5671.398,E2 -5671.398} C_VEL
LIN {X 0,Y 503.633,Z 475.748,A -85,B 0,C 180,E1 -5672.199,E2 -5672.199} C_VEL
LIN {X 0,Y 503.32,Z 485.987,A -85,B 0,C 180,E1 -5673.101,E2 -5673.101} C_VEL
LIN {X 0,Y 502.982,Z 494.405,A -85,B 0,C 180,E1 -5674.005,E2 -5674.005} C_VEL
LIN {X 0,Y 502.733,Z 502.174,A -85,B 0,C 180,E1 -5675.012,E2 -5675.012} C_VEL
LIN {X 0,Y 502.533,Z 509.777,A -85,B 0,C 180,E1 -5676.221,E2 -5676.221} C_VEL
LIN {X 0,Y 502.327,Z 516.817,A -85,B 0,C 180,E1 -5677.637,E2 -5677.637} C_VEL
LIN {X 0,Y 502.186,Z 521.511,A -85,B 0,C 180,E1 -5678.855,E2 -5678.855} C_VEL
LIN {X 0,Y 502.161,Z 525.093,A -85,B 0,C 180,E1 -5680.075,E2 -5680.075} C_VEL
LIN {X 0,Y 502.097,Z 528.058,A -85,B 0,C 180,E1 -5681.533,E2 -5681.533} C_VEL
LIN {X 0,Y 501.995,Z 529.612,A -85,B 0,C 180,E1 -5682.943,E2 -5682.943} C_VEL
LIN {X 0,Y 502.012,Z 529.956,A -85,B 0,C 180,E1 -5683.767,E2 -5683.767} C_VEL
LIN {X 0,Y 502.046,Z 529.699,A -85,B 0,C 180,E1 -5685.004,E2 -5685.004} C_VEL
LIN {X 0,Y 501.995,Z 528.48,A -85,B 0,C 180,E1 -5686.259,E2 -5686.259} C_VEL
LIN {X 0,Y 502.044,Z 527.127,A -85,B 0,C 180,E1 -5687.095,E2 -5687.095} C_VEL
LIN {X 0,Y 502.126,Z 524.215,A -85,B 0,C 180,E1 -5688.355,E2 -5688.355} C_VEL
LIN {X 0,Y 502.247,Z 520.168,A -85,B 0,C 180,E1 -5689.622,E2 -5689.622} C_VEL
LIN {X 0,Y 502.358,Z 514.84,A -85,B 0,C 180,E1 -5690.9,E2 -5690.9} C_VEL
LIN {X 0,Y 502.592,Z 507.986,A -85,B 0,C 180,E1 -5692.181,E2 -5692.181} C_VEL
LIN {X 0,Y 502.867,Z 499.324,A -85,B 0,C 180,E1 -5693.472,E2 -5693.472} C_VEL
LIN {X 0,Y 503.184,Z 490.29,A -85,B 0,C 180,E1 -5694.551,E2 -5694.551} C_VEL
LIN {X 0,Y 503.489,Z 480.297,A -85,B 0,C 180,E1 -5695.517,E2 -5695.517} C_VEL
LIN {X 0,Y 503.876,Z 468.978,A -85,B 0,C 180,E1 -5696.396,E2 -5696.396} C_VEL
LIN {X 0,Y 504.256,Z 457.086,A -85,B 0,C 180,E1 -5697.115,E2 -5697.115} C_VEL
LIN {X 0,Y 504.531,Z 445.499,A -85,B 0,C 180,E1 -5697.647,E2 -5697.647} C_VEL
LIN {X 0,Y 504.752,Z 433.084,A -85,B 0,C 180,E1 -5698.057,E2 -5698.057} C_VEL
LIN {X 0,Y 504.921,Z 420.34,A -85,B 0,C 180,E1 -5698.319,E2 -5698.319} C_VEL
LIN {X 0,Y 505.352,Z 330.463,A -85,B 0,C 180,E1 -5699.608,E2 -5699.608} C_VEL
LIN {X 0,Y 503.265,Z 319.069,A -85,B 0,C 180,E1 -5699.853,E2 -5699.853} C_VEL
LIN {X 0,Y 503.529,Z 302.007,A -85,B 0,C 180,E1 -5702.979,E2 -5702.979} C_VEL
LIN {X 0,Y 503.467,Z 296.79,A -85,B 0,C 180,E1 -5703.942,E2 -5703.942} C_VEL
LIN {X 0,Y 502.837,Z 292.853,A -85,B 0,C 180,E1 -5704.714,E2 -5704.714} C_VEL
LIN {X 0,Y 502.786,Z 292.854,A -85,B 0,C 180,E1 -5707.953,E2 -5707.953} C_VEL
LIN {X 0,Y 502.77,Z 292.859,A -85,B 0,C 180,E1 -5711.069,E2 -5711.069} C_VEL
LIN {X 0,Y 502.749,Z 292.861,A -85,B 0,C 180,E1 -5713.372,E2 -5713.372} C_VEL
LIN {X 0,Y 502.771,Z 292.855,A -85,B 0,C 180,E1 -5715.659,E2 -5715.659} C_VEL
LIN {X 0,Y 502.762,Z 292.86,A -85,B 0,C 180,E1 -5719.011,E2 -5719.011} C_VEL
LIN {X 0,Y 502.783,Z 292.851,A -85,B 0,C 180,E1 -5722.045,E2 -5722.045} C_VEL
LIN {X 0,Y 502.787,Z 292.855,A -85,B 0,C 180,E1 -5725.033,E2 -5725.033} C_VEL
LIN {X 0,Y 502.773,Z 292.856,A -85,B 0,C 180,E1 -5727.915,E2 -5727.915} C_VEL
LIN {X 0,Y 502.802,Z 292.847,A -85,B 0,C 180,E1 -5730.711,E2 -5730.711} C_VEL
LIN {X 0,Y 502.762,Z 292.861,A -85,B 0,C 180,E1 -5733.46,E2 -5733.46} C_VEL
LIN {X 0,Y 502.757,Z 292.858,A -85,B 0,C 180,E1 -5736.085,E2 -5736.085} C_VEL
LIN {X 0,Y 502.771,Z 292.851,A -85,B 0,C 180,E1 -5738.688,E2 -5738.688} C_VEL
LIN {X 0,Y 502.8,Z 292.85,A -85,B 0,C 180,E1 -5741.247,E2 -5741.247} C_VEL
LIN {X 0,Y 502.825,Z 292.846,A -85,B 0,C 180,E1 -5744.665,E2 -5744.665} C_VEL
LIN {X 0,Y 502.859,Z 292.847,A -85,B 0,C 180,E1 -5748.043,E2 -5748.043} C_VEL
LIN {X 0,Y 502.824,Z 292.842,A -85,B 0,C 180,E1 -5751.156,E2 -5751.156} C_VEL
LIN {X 0,Y 502.837,Z 292.844,A -85,B 0,C 180,E1 -5753.58,E2 -5753.58} C_VEL
LIN {X 0,Y 502.732,Z 292.86,A -85,B 0,C 180,E1 -5755.992,E2 -5755.992} C_VEL
LIN {X 0,Y 502.992,Z 292.822,A -85,B 0,C 180,E1 -5757.598,E2 -5757.598} C_VEL
LIN {X 0,Y 502.978,Z 292.828,A -85,B 0,C 180,E1 -5760.801,E2 -5760.801} C_VEL
LIN {X 0,Y 502.994,Z 292.828,A -85,B 0,C 180,E1 -5762.403,E2 -5762.403} C_VEL
LIN {X 0,Y 502.907,Z 292.835,A -85,B 0,C 180,E1 -5765.614,E2 -5765.614} C_VEL
LIN {X 0,Y 502.844,Z 292.839,A -85,B 0,C 180,E1 -5768.034,E2 -5768.034} C_VEL
LIN {X 0,Y 502.863,Z 292.841,A -85,B 0,C 180,E1 -5771.284,E2 -5771.284} C_VEL
LIN {X 0,Y 502.815,Z 292.848,A -85,B 0,C 180,E1 -5774.572,E2 -5774.572} C_VEL
LIN {X 0,Y 502.808,Z 292.843,A -85,B 0,C 180,E1 -5777.909,E2 -5777.909} C_VEL
LIN {X 0,Y 502.821,Z 292.847,A -85,B 0,C 180,E1 -5780.537,E2 -5780.537} C_VEL
LIN {X 0,Y 502.778,Z 292.856,A -85,B 0,C 180,E1 -5783.041,E2 -5783.041} C_VEL
LIN {X 0,Y 502.771,Z 292.855,A -85,B 0,C 180,E1 -5785.68,E2 -5785.68} C_VEL
LIN {X 0,Y 502.788,Z 292.849,A -85,B 0,C 180,E1 -5788.376,E2 -5788.376} C_VEL
LIN {X 0,Y 502.786,Z 292.856,A -85,B 0,C 180,E1 -5791.144,E2 -5791.144} C_VEL
LIN {X 0,Y 502.796,Z 292.851,A -85,B 0,C 180,E1 -5793.995,E2 -5793.995} C_VEL
LIN {X 0,Y 502.758,Z 292.858,A -85,B 0,C 180,E1 -5797.177,E2 -5797.177} C_VEL
LIN {X 0,Y 502.767,Z 292.858,A -85,B 0,C 180,E1 -5800.017,E2 -5800.017} C_VEL
LIN {X 0,Y 502.798,Z 292.848,A -85,B 0,C 180,E1 -5802.2,E2 -5802.2} C_VEL
LIN {X 0,Y 502.781,Z 292.855,A -85,B 0,C 180,E1 -5805.471,E2 -5805.471} C_VEL
LIN {X 0,Y 502.79,Z 292.859,A -85,B 0,C 180,E1 -5807.861,E2 -5807.861} C_VEL
LIN {X 0,Y 502.797,Z 292.851,A -85,B 0,C 180,E1 -5811.025,E2 -5811.025} C_VEL
LIN {X 0,Y 502.768,Z 292.86,A -85,B 0,C 180,E1 -5814.171,E2 -5814.171} C_VEL
LIN {X 0,Y 502.83,Z 292.847,A -85,B 0,C 180,E1 -5816.994,E2 -5816.994} C_VEL
LIN {X 0,Y 502.812,Z 292.854,A -85,B 0,C 180,E1 -5820.066,E2 -5820.066} C_VEL
LIN {X 0,Y 502.822,Z 292.855,A -85,B 0,C 180,E1 -5822.534,E2 -5822.534} C_VEL
LIN {X 0,Y 502.807,Z 292.97,A -85,B 0,C 180,E1 -5825.397,E2 -5825.397} C_VEL
LIN {X 0,Y 504.455,Z 302.12,A -85,B 0,C 180,E1 -5827.041,E2 -5827.041} C_VEL
LIN {X 0,Y 504.009,Z 317.42,A -85,B 0,C 180,E1 -5829.599,E2 -5829.599} C_VEL
LIN {X 0,Y 503.534,Z 334.006,A -85,B 0,C 180,E1 -5832.329,E2 -5832.329} C_VEL
LIN {X 0,Y 503.296,Z 345.696,A -85,B 0,C 180,E1 -5834.199,E2 -5834.199} C_VEL
LIN {X 0,Y 505.406,Z 359.46,A -85,B 0,C 180,E1 -5834.466,E2 -5834.466} C_VEL
LIN {X 0,Y 504.893,Z 453.396,A -85,B 0,C 180,E1 -5835.825,E2 -5835.825} C_VEL
LIN {X 0,Y 504.591,Z 465.995,A -85,B 0,C 180,E1 -5836.15,E2 -5836.15} C_VEL
LIN {X 0,Y 504.277,Z 478.972,A -85,B 0,C 180,E1 -5836.655,E2 -5836.655} C_VEL
LIN {X 0,Y 503.959,Z 490.954,A -85,B 0,C 180,E1 -5837.291,E2 -5837.291} C_VEL
LIN {X 0,Y 503.617,Z 501.621,A -85,B 0,C 180,E1 -5838.02,E2 -5838.02} C_VEL
LIN {X 0,Y 503.249,Z 512.307,A -85,B 0,C 180,E1 -5838.93,E2 -5838.93} C_VEL
LIN {X 0,Y 502.909,Z 521.937,A -85,B 0,C 180,E1 -5839.941,E2 -5839.941} C_VEL
LIN {X 0,Y 502.65,Z 529.831,A -85,B 0,C 180,E1 -5840.951,E2 -5840.951} C_VEL
LIN {X 0,Y 502.401,Z 537.541,A -85,B 0,C 180,E1 -5842.162,E2 -5842.162} C_VEL
LIN {X 0,Y 502.236,Z 544.238,A -85,B 0,C 180,E1 -5843.483,E2 -5843.483} C_VEL
LIN {X 0,Y 502.174,Z 549.376,A -85,B 0,C 180,E1 -5844.781,E2 -5844.781} C_VEL
LIN {X 0,Y 502.138,Z 552.99,A -85,B 0,C 180,E1 -5845.988,E2 -5845.988} C_VEL
LIN {X 0,Y 502.12,Z 554.853,A -85,B 0,C 180,E1 -5846.791,E2 -5846.791} C_VEL
LIN {X 0,Y 502.091,Z 556.251,A -85,B 0,C 180,E1 -5847.594,E2 -5847.594} C_VEL
LIN {X 0,Y 501.99,Z 557.856,A -85,B 0,C 180,E1 -5849.199,E2 -5849.199} C_VEL
LIN {X 0,Y 501.981,Z 558.073,A -85,B 0,C 180,E1 -5850.001,E2 -5850.001} C_VEL
LIN {X 0,Y 502.036,Z 557.253,A -85,B 0,C 180,E1 -5851.605,E2 -5851.605} C_VEL
LIN {X 0,Y 502.091,Z 556.26,A -85,B 0,C 180,E1 -5852.407,E2 -5852.407} C_VEL
LIN {X 0,Y 502.121,Z 554.865,A -85,B 0,C 180,E1 -5853.21,E2 -5853.21} C_VEL
LIN {X 0,Y 502.102,Z 551.929,A -85,B 0,C 180,E1 -5854.416,E2 -5854.416} C_VEL
LIN {X 0,Y 502.21,Z 547.956,A -85,B 0,C 180,E1 -5855.622,E2 -5855.622} C_VEL
LIN {X 0,Y 502.329,Z 541.943,A -85,B 0,C 180,E1 -5857.012,E2 -5857.012} C_VEL
LIN {X 0,Y 502.478,Z 535.16,A -85,B 0,C 180,E1 -5858.243,E2 -5858.243} C_VEL
LIN {X 0,Y 502.747,Z 526.871,A -85,B 0,C 180,E1 -5859.455,E2 -5859.455} C_VEL
LIN {X 0,Y 502.991,Z 518.37,A -85,B 0,C 180,E1 -5860.466,E2 -5860.466} C_VEL
LIN {X 0,Y 503.412,Z 507.869,A -85,B 0,C 180,E1 -5861.476,E2 -5861.476} C_VEL
LIN {X 0,Y 503.711,Z 496.283,A -85,B 0,C 180,E1 -5862.371,E2 -5862.371} C_VEL
LIN {X 0,Y 504.133,Z 484.144,A -85,B 0,C 180,E1 -5863.094,E2 -5863.094} C_VEL
LIN {X 0,Y 504.514,Z 471.762,A -85,B 0,C 180,E1 -5863.648,E2 -5863.648} C_VEL
LIN {X 0,Y 504.754,Z 459.949,A -85,B 0,C 180,E1 -5864.026,E2 -5864.026} C_VEL
LIN {X 0,Y 504.952,Z 447.405,A -85,B 0,C 180,E1 -5864.278,E2 -5864.278} C_VEL
LIN {X 0,Y 505.212,Z 357.992,A -85,B 0,C 180,E1 -5865.562,E2 -5865.562} C_VEL
LIN {X 0,Y 503.259,Z 345.439,A -85,B 0,C 180,E1 -5865.825,E2 -5865.825} C_VEL
LIN {X 0,Y 503.806,Z 326.522,A -85,B 0,C 180,E1 -5868.926,E2 -5868.926} C_VEL
LIN {X 0,Y 504.375,Z 307.416,A -85,B 0,C 180,E1 -5872.1,E2 -5872.1} C_VEL
LIN {X 0,Y 504.421,Z 301.273,A -85,B 0,C 180,E1 -5873.137,E2 -5873.137} C_VEL
LIN {X 0,Y 502.809,Z 292.853,A -85,B 0,C 180,E1 -5874.657,E2 -5874.657} C_VEL
LIN {X 0,Y 502.828,Z 292.854,A -85,B 0,C 180,E1 -5877.468,E2 -5877.468} C_VEL
LIN {X 0,Y 502.812,Z 292.85,A -85,B 0,C 180,E1 -5880.212,E2 -5880.212} C_VEL
LIN {X 0,Y 502.836,Z 292.844,A -85,B 0,C 180,E1 -5883.032,E2 -5883.032} C_VEL
LIN {X 0,Y 502.771,Z 292.86,A -85,B 0,C 180,E1 -5885.952,E2 -5885.952} C_VEL
LIN {X 0,Y 502.797,Z 292.849,A -85,B 0,C 180,E1 -5888.977,E2 -5888.977} C_VEL
LIN {X 0,Y 502.807,Z 292.856,A -85,B 0,C 180,E1 -5892.199,E2 -5892.199} C_VEL
LIN {X 0,Y 502.789,Z 292.849,A -85,B 0,C 180,E1 -5895.47,E2 -5895.47} C_VEL
LIN {X 0,Y 502.799,Z 292.849,A -85,B 0,C 180,E1 -5897.861,E2 -5897.861} C_VEL
LIN {X 0,Y 502.804,Z 292.851,A -85,B 0,C 180,E1 -5901.024,E2 -5901.024} C_VEL
LIN {X 0,Y 502.775,Z 292.853,A -85,B 0,C 180,E1 -5904.17,E2 -5904.17} C_VEL
LIN {X 0,Y 502.837,Z 292.851,A -85,B 0,C 180,E1 -5906.993,E2 -5906.993} C_VEL
LIN {X 0,Y 502.818,Z 292.846,A -85,B 0,C 180,E1 -5910.065,E2 -5910.065} C_VEL
LIN {X 0,Y 502.847,Z 292.846,A -85,B 0,C 180,E1 -5913.444,E2 -5913.444} C_VEL
LIN {X 0,Y 502.79,Z 292.855,A -85,B 0,C 180,E1 -5916.959,E2 -5916.959} C_VEL
LIN {X 0,Y 502.84,Z 292.849,A -85,B 0,C 180,E1 -5919.548,E2 -5919.548} C_VEL
LIN {X 0,Y 502.826,Z 292.846,A -85,B 0,C 180,E1 -5922.092,E2 -5922.092} C_VEL
LIN {X 0,Y 502.846,Z 292.85,A -85,B 0,C 180,E1 -5925.429,E2 -5925.429} C_VEL
LIN {X 0,Y 502.879,Z 292.838,A -85,B 0,C 180,E1 -5928.717,E2 -5928.717} C_VEL
LIN {X 0,Y 502.877,Z 292.845,A -85,B 0,C 180,E1 -5931.966,E2 -5931.966} C_VEL
LIN {X 0,Y 502.931,Z 292.834,A -85,B 0,C 180,E1 -5934.386,E2 -5934.386} C_VEL
LIN {X 0,Y 503.021,Z 292.824,A -85,B 0,C 180,E1 -5937.598,E2 -5937.598} C_VEL
LIN {X 0,Y 503.03,Z 292.827,A -85,B 0,C 180,E1 -5940,E2 -5940} C_VEL
LIN {X 0,Y 503.02,Z 292.827,A -85,B 0,C 180,E1 -5942.402,E2 -5942.402} C_VEL
LIN {X 0,Y 502.919,Z 292.834,A -85,B 0,C 180,E1 -5945.614,E2 -5945.614} C_VEL
LIN {X 0,Y 502.871,Z 292.843,A -85,B 0,C 180,E1 -5948.843,E2 -5948.843} C_VEL
LIN {X 0,Y 502.848,Z 292.845,A -85,B 0,C 180,E1 -5952.101,E2 -5952.101} C_VEL
LIN {X 0,Y 502.852,Z 292.842,A -85,B 0,C 180,E1 -5955.399,E2 -5955.399} C_VEL
LIN {X 0,Y 502.828,Z 292.853,A -85,B 0,C 180,E1 -5958.752,E2 -5958.752} C_VEL
LIN {X 0,Y 502.786,Z 292.854,A -85,B 0,C 180,E1 -5961.311,E2 -5961.311} C_VEL
LIN {X 0,Y 502.775,Z 292.851,A -85,B 0,C 180,E1 -5963.914,E2 -5963.914} C_VEL
LIN {X 0,Y 502.838,Z 292.845,A -85,B 0,C 180,E1 -5966.567,E2 -5966.567} C_VEL
LIN {X 0,Y 502.816,Z 292.847,A -85,B 0,C 180,E1 -5969.935,E2 -5969.935} C_VEL
LIN {X 0,Y 502.831,Z 292.848,A -85,B 0,C 180,E1 -5973.031,E2 -5973.031} C_VEL
LIN {X 0,Y 502.77,Z 292.855,A -85,B 0,C 180,E1 -5975.951,E2 -5975.951} C_VEL
LIN {X 0,Y 502.803,Z 292.849,A -85,B 0,C 180,E1 -5978.976,E2 -5978.976} C_VEL
LIN {X 0,Y 502.805,Z 292.85,A -85,B 0,C 180,E1 -5982.199,E2 -5982.199} C_VEL
LIN {X 0,Y 502.787,Z 292.853,A -85,B 0,C 180,E1 -5985.47,E2 -5985.47} C_VEL
LIN {X 0,Y 502.796,Z 292.857,A -85,B 0,C 180,E1 -5987.86,E2 -5987.86} C_VEL
LIN {X 0,Y 502.797,Z 292.848,A -85,B 0,C 180,E1 -5991.023,E2 -5991.023} C_VEL
LIN {X 0,Y 502.773,Z 292.861,A -85,B 0,C 180,E1 -5994.169,E2 -5994.169} C_VEL
LIN {X 0,Y 502.811,Z 292.847,A -85,B 0,C 180,E1 -5997.213,E2 -5997.213} C_VEL
LIN {X 0,Y 502.11,Z 292.939,A -85,B 0,C 180,E1 -5997.882,E2 -5997.882} C_VEL
LIN {X 0,Y 499.248,Z 293.294,A -85,B 0,C 180,E1 -5998.968,E2 -5998.968} C_VEL
LIN {X 0,Y 496.85,Z 293.594,A -85,B 0,C 180,E1 -5999.842,E2 -5999.842} C_VEL
LIN {X 0,Y 495.822,Z 293.726,A -85,B 0,C 180,E1 -6000.518,E2 -6000.518} C_VEL
LIN {X 0,Y 495.739,Z 293.729,A -85,B 0,C 180,E1 -6000.747,E2 -6000.747} C_VEL
LIN {X 0,Y 495.755,Z 293.727,A -85,B 0,C 180,E1 -6003.93,E2 -6003.93} C_VEL
LIN {X 0,Y 495.759,Z 293.728,A -85,B 0,C 180,E1 -6007.139,E2 -6007.139} C_VEL
LIN {X 0,Y 495.768,Z 293.725,A -85,B 0,C 180,E1 -6010.109,E2 -6010.109} C_VEL
LIN {X 0,Y 495.758,Z 293.731,A -85,B 0,C 180,E1 -6012.68,E2 -6012.68} C_VEL
LIN {X 0,Y 495.787,Z 293.728,A -85,B 0,C 180,E1 -6015.216,E2 -6015.216} C_VEL
LIN {X 0,Y 495.85,Z 293.716,A -85,B 0,C 180,E1 -6018.554,E2 -6018.554} C_VEL
LIN {X 0,Y 495.836,Z 293.722,A -85,B 0,C 180,E1 -6021.851,E2 -6021.851} C_VEL
LIN {X 0,Y 495.906,Z 293.899,A -85,B 0,C 180,E1 -6023.072,E2 -6023.072} C_VEL
LIN {X 0,Y 496.692,Z 299.046,A -85,B 0,C 180,E1 -6024.111,E2 -6024.111} C_VEL
LIN {X 0,Y 496.41,Z 312.757,A -85,B 0,C 180,E1 -6026.753,E2 -6026.753} C_VEL
LIN {X 0,Y 496.316,Z 319.652,A -85,B 0,C 180,E1 -6028.034,E2 -6028.034} C_VEL
LIN {X 0,Y 498.574,Z 331.484,A -85,B 0,C 180,E1 -6028.283,E2 -6028.283} C_VEL
LIN {X 0,Y 498.018,Z 427.204,A -85,B 0,C 180,E1 -6029.696,E2 -6029.696} C_VEL
LIN {X 0,Y 497.751,Z 440.106,A -85,B 0,C 180,E1 -6030.05,E2 -6030.05} C_VEL
LIN {X 0,Y 497.464,Z 452.564,A -85,B 0,C 180,E1 -6030.556,E2 -6030.556} C_VEL
LIN {X 0,Y 497.1,Z 464.485,A -85,B 0,C 180,E1 -6031.214,E2 -6031.214} C_VEL
LIN {X 0,Y 496.692,Z 475.87,A -85,B 0,C 180,E1 -6032.026,E2 -6032.026} C_VEL
LIN {X 0,Y 496.352,Z 486.131,A -85,B 0,C 180,E1 -6032.941,E2 -6032.941} C_VEL
LIN {X 0,Y 495.986,Z 494.561,A -85,B 0,C 180,E1 -6033.859,E2 -6033.859} C_VEL
LIN {X 0,Y 495.652,Z 503.703,A -85,B 0,C 180,E1 -6035.083,E2 -6035.083} C_VEL
LIN {X 0,Y 495.45,Z 511.063,A -85,B 0,C 180,E1 -6036.311,E2 -6036.311} C_VEL
LIN {X 0,Y 495.246,Z 517.869,A -85,B 0,C 180,E1 -6037.747,E2 -6037.747} C_VEL
LIN {X 0,Y 495.105,Z 522.368,A -85,B 0,C 180,E1 -6038.982,E2 -6038.982} C_VEL
LIN {X 0,Y 495.054,Z 524.745,A -85,B 0,C 180,E1 -6039.808,E2 -6039.808} C_VEL
LIN {X 0,Y 495.014,Z 526.692,A -85,B 0,C 180,E1 -6040.635,E2 -6040.635} C_VEL
LIN {X 0,Y 495.004,Z 528.366,A -85,B 0,C 180,E1 -6041.579,E2 -6041.579} C_VEL
LIN {X 0,Y 494.919,Z 529.93,A -85,B 0,C 180,E1 -6043.132,E2 -6043.132} C_VEL
LIN {X 0,Y 494.923,Z 530.195,A -85,B 0,C 180,E1 -6043.968,E2 -6043.968} C_VEL
LIN {X 0,Y 494.958,Z 529.858,A -85,B 0,C 180,E1 -6045.085,E2 -6045.085} C_VEL
LIN {X 0,Y 494.905,Z 528.395,A -85,B 0,C 180,E1 -6046.499,E2 -6046.499} C_VEL
LIN {X 0,Y 495.06,Z 525.535,A -85,B 0,C 180,E1 -6047.983,E2 -6047.983} C_VEL
LIN {X 0,Y 495.16,Z 521.126,A -85,B 0,C 180,E1 -6049.483,E2 -6049.483} C_VEL
LIN {X 0,Y 495.29,Z 515.055,A -85,B 0,C 180,E1 -6050.994,E2 -6050.994} C_VEL
LIN {X 0,Y 495.552,Z 508.205,A -85,B 0,C 180,E1 -6052.294,E2 -6052.294} C_VEL
LIN {X 0,Y 495.842,Z 499.546,A -85,B 0,C 180,E1 -6053.603,E2 -6053.603} C_VEL
LIN {X 0,Y 496.197,Z 490.796,A -85,B 0,C 180,E1 -6054.668,E2 -6054.668} C_VEL
LIN {X 0,Y 496.525,Z 480.427,A -85,B 0,C 180,E1 -6055.687,E2 -6055.687} C_VEL
LIN {X 0,Y 496.948,Z 469.263,A -85,B 0,C 180,E1 -6056.566,E2 -6056.566} C_VEL
LIN {X 0,Y 497.332,Z 457.931,A -85,B 0,C 180,E1 -6057.268,E2 -6057.268} C_VEL
LIN {X 0,Y 497.644,Z 445.887,A -85,B 0,C 180,E1 -6057.834,E2 -6057.834} C_VEL
LIN {X 0,Y 497.886,Z 432.569,A -85,B 0,C 180,E1 -6058.277,E2 -6058.277} C_VEL
LIN {X 0,Y 498.059,Z 418.443,A -85,B 0,C 180,E1 -6058.554,E2 -6058.554} C_VEL
LIN {X 0,Y 498.586,Z 331.486,A -85,B 0,C 180,E1 -6059.816,E2 -6059.816} C_VEL
LIN {X 0,Y 496.276,Z 319.222,A -85,B 0,C 180,E1 -6060.089,E2 -6060.089} C_VEL
LIN {X 0,Y 496.629,Z 302.418,A -85,B 0,C 180,E1 -6063.202,E2 -6063.202} C_VEL
LIN {X 0,Y 496.316,Z 296.84,A -85,B 0,C 180,E1 -6064.254,E2 -6064.254} C_VEL
LIN {X 0,Y 495.771,Z 293.733,A -85,B 0,C 180,E1 -6064.881,E2 -6064.881} C_VEL
LIN {X 0,Y 495.722,Z 293.735,A -85,B 0,C 180,E1 -6067.561,E2 -6067.561} C_VEL
LIN {X 0,Y 495.738,Z 293.731,A -85,B 0,C 180,E1 -6070.044,E2 -6070.044} C_VEL
LIN {X 0,Y 495.708,Z 293.74,A -85,B 0,C 180,E1 -6072.884,E2 -6072.884} C_VEL
LIN {X 0,Y 495.715,Z 293.733,A -85,B 0,C 180,E1 -6075.997,E2 -6075.997} C_VEL
LIN {X 0,Y 495.722,Z 293.738,A -85,B 0,C 180,E1 -6079.296,E2 -6079.296} C_VEL
LIN {X 0,Y 495.737,Z 293.736,A -85,B 0,C 180,E1 -6081.407,E2 -6081.407} C_VEL
LIN {X 0,Y 495.738,Z 293.729,A -85,B 0,C 180,E1 -6084.462,E2 -6084.462} C_VEL
LIN {X 0,Y 495.743,Z 293.729,A -85,B 0,C 180,E1 -6087.404,E2 -6087.404} C_VEL
LIN {X 0,Y 495.753,Z 293.726,A -85,B 0,C 180,E1 -6090.253,E2 -6090.253} C_VEL
LIN {X 0,Y 495.728,Z 293.734,A -85,B 0,C 180,E1 -6093.27,E2 -6093.27} C_VEL
LIN {X 0,Y 495.729,Z 293.73,A -85,B 0,C 180,E1 -6096.612,E2 -6096.612} C_VEL
LIN {X 0,Y 495.77,Z 293.726,A -85,B 0,C 180,E1 -6099.324,E2 -6099.324} C_VEL
LIN {X 0,Y 495.769,Z 293.73,A -85,B 0,C 180,E1 -6101.828,E2 -6101.828} C_VEL
LIN {X 0,Y 495.765,Z 293.725,A -85,B 0,C 180,E1 -6105.217,E2 -6105.217} C_VEL
LIN {X 0,Y 495.811,Z 293.722,A -85,B 0,C 180,E1 -6108.554,E2 -6108.554} C_VEL
LIN {X 0,Y 495.799,Z 293.721,A -85,B 0,C 180,E1 -6111.851,E2 -6111.851} C_VEL
LIN {X 0,Y 495.831,Z 293.725,A -85,B 0,C 180,E1 -6114.306,E2 -6114.306} C_VEL
LIN {X 0,Y 495.959,Z 293.698,A -85,B 0,C 180,E1 -6117.564,E2 -6117.564} C_VEL
LIN {X 0,Y 495.93,Z 293.706,A -85,B 0,C 180,E1 -6120.812,E2 -6120.812} C_VEL
LIN {X 0,Y 495.961,Z 293.703,A -85,B 0,C 180,E1 -6122.437,E2 -6122.437} C_VEL
LIN {X 0,Y 495.863,Z 293.713,A -85,B 0,C 180,E1 -6125.694,E2 -6125.694} C_VEL
LIN {X 0,Y 495.806,Z 293.717,A -85,B 0,C 180,E1 -6128.149,E2 -6128.149} C_VEL
LIN {X 0,Y 495.839,Z 293.715,A -85,B 0,C 180,E1 -6131.446,E2 -6131.446} C_VEL
LIN {X 0,Y 495.767,Z 293.729,A -85,B 0,C 180,E1 -6134.784,E2 -6134.784} C_VEL
LIN {X 0,Y 495.771,Z 293.72,A -85,B 0,C 180,E1 -6138.172,E2 -6138.172} C_VEL
LIN {X 0,Y 495.766,Z 293.728,A -85,B 0,C 180,E1 -6140.757,E2 -6140.757} C_VEL
LIN {X 0,Y 495.73,Z 293.734,A -85,B 0,C 180,E1 -6143.388,E2 -6143.388} C_VEL
LIN {X 0,Y 495.732,Z 293.731,A -85,B 0,C 180,E1 -6146.731,E2 -6146.731} C_VEL
LIN {X 0,Y 495.755,Z 293.73,A -85,B 0,C 180,E1 -6149.747,E2 -6149.747} C_VEL
LIN {X 0,Y 495.761,Z 293.725,A -85,B 0,C 180,E1 -6152.595,E2 -6152.595} C_VEL
LIN {X 0,Y 495.738,Z 293.734,A -85,B 0,C 180,E1 -6155.539,E2 -6155.539} C_VEL
LIN {X 0,Y 495.752,Z 293.726,A -85,B 0,C 180,E1 -6158.768,E2 -6158.768} C_VEL
LIN {X 0,Y 495.739,Z 293.733,A -85,B 0,C 180,E1 -6161.783,E2 -6161.783} C_VEL
LIN {X 0,Y 495.732,Z 293.73,A -85,B 0,C 180,E1 -6165.142,E2 -6165.142} C_VEL
LIN {X 0,Y 495.746,Z 293.735,A -85,B 0,C 180,E1 -6168.219,E2 -6168.219} C_VEL
LIN {X 0,Y 495.745,Z 293.731,A -85,B 0,C 180,E1 -6171.409,E2 -6171.409} C_VEL
LIN {X 0,Y 495.742,Z 293.731,A -85,B 0,C 180,E1 -6174.463,E2 -6174.463} C_VEL
LIN {X 0,Y 495.765,Z 293.727,A -85,B 0,C 180,E1 -6177.407,E2 -6177.407} C_VEL
LIN {X 0,Y 495.763,Z 293.732,A -85,B 0,C 180,E1 -6180.255,E2 -6180.255} C_VEL
LIN {X 0,Y 495.804,Z 293.725,A -85,B 0,C 180,E1 -6183.256,E2 -6183.256} C_VEL
LIN {X 0,Y 495.759,Z 293.787,A -85,B 0,C 180,E1 -6185.187,E2 -6185.187} C_VEL
LIN {X 0,Y 497.466,Z 302.842,A -85,B 0,C 180,E1 -6186.848,E2 -6186.848} C_VEL
LIN {X 0,Y 497.238,Z 313.928,A -85,B 0,C 180,E1 -6188.738,E2 -6188.738} C_VEL
LIN {X 0,Y 496.584,Z 333.833,A -85,B 0,C 180,E1 -6192.073,E2 -6192.073} C_VEL
LIN {X 0,Y 496.252,Z 345.207,A -85,B 0,C 180,E1 -6193.955,E2 -6193.955} C_VEL
LIN {X 0,Y 498.556,Z 360.795,A -85,B 0,C 180,E1 -6194.267,E2 -6194.267} C_VEL
LIN {X 0,Y 498.032,Z 453.273,A -85,B 0,C 180,E1 -6195.625,E2 -6195.625} C_VEL
LIN {X 0,Y 497.693,Z 465.832,A -85,B 0,C 180,E1 -6195.954,E2 -6195.954} C_VEL
LIN {X 0,Y 497.374,Z 478.786,A -85,B 0,C 180,E1 -6196.466,E2 -6196.466} C_VEL
LIN {X 0,Y 497.019,Z 491.054,A -85,B 0,C 180,E1 -6197.13,E2 -6197.13} C_VEL
LIN {X 0,Y 496.621,Z 502.704,A -85,B 0,C 180,E1 -6197.953,E2 -6197.953} C_VEL
LIN {X 0,Y 496.222,Z 513.167,A -85,B 0,C 180,E1 -6198.875,E2 -6198.875} C_VEL
LIN {X 0,Y 495.861,Z 521.725,A -85,B 0,C 180,E1 -6199.796,E2 -6199.796} C_VEL
LIN {X 0,Y 495.617,Z 529.622,A -85,B 0,C 180,E1 -6200.821,E2 -6200.821} C_VEL
LIN {X 0,Y 495.342,Z 537.334,A -85,B 0,C 180,E1 -6202.049,E2 -6202.049} C_VEL
LIN {X 0,Y 495.164,Z 544.443,A -85,B 0,C 180,E1 -6203.481,E2 -6203.481} C_VEL
LIN {X 0,Y 495.106,Z 549.174,A -85,B 0,C 180,E1 -6204.707,E2 -6204.707} C_VEL
LIN {X 0,Y 495.032,Z 552.788,A -85,B 0,C 180,E1 -6205.93,E2 -6205.93} C_VEL
LIN {X 0,Y 495.042,Z 554.653,A -85,B 0,C 180,E1 -6206.745,E2 -6206.745} C_VEL
LIN {X 0,Y 494.997,Z 556.051,A -85,B 0,C 180,E1 -6207.56,E2 -6207.56} C_VEL
LIN {X 0,Y 494.962,Z 557.048,A -85,B 0,C 180,E1 -6208.373,E2 -6208.373} C_VEL
LIN {X 0,Y 494.899,Z 557.875,A -85,B 0,C 180,E1 -6210.001,E2 -6210.001} C_VEL
LIN {X 0,Y 494.962,Z 557.056,A -85,B 0,C 180,E1 -6211.628,E2 -6211.628} C_VEL
LIN {X 0,Y 494.998,Z 556.062,A -85,B 0,C 180,E1 -6212.442,E2 -6212.442} C_VEL
LIN {X 0,Y 495.042,Z 554.667,A -85,B 0,C 180,E1 -6213.256,E2 -6213.256} C_VEL
LIN {X 0,Y 495.008,Z 551.73,A -85,B 0,C 180,E1 -6214.479,E2 -6214.479} C_VEL
LIN {X 0,Y 495.127,Z 547.757,A -85,B 0,C 180,E1 -6215.703,E2 -6215.703} C_VEL
LIN {X 0,Y 495.255,Z 541.641,A -85,B 0,C 180,E1 -6217.133,E2 -6217.133} C_VEL
LIN {X 0,Y 495.425,Z 534.959,A -85,B 0,C 180,E1 -6218.361,E2 -6218.361} C_VEL
LIN {X 0,Y 495.717,Z 526.668,A -85,B 0,C 180,E1 -6219.59,E2 -6219.59} C_VEL
LIN {X 0,Y 495.984,Z 518.165,A -85,B 0,C 180,E1 -6220.616,E2 -6220.616} C_VEL
LIN {X 0,Y 496.429,Z 507.662,A -85,B 0,C 180,E1 -6221.639,E2 -6221.639} C_VEL
LIN {X 0,Y 496.761,Z 496.338,A -85,B 0,C 180,E1 -6222.528,E2 -6222.528} C_VEL
LIN {X 0,Y 497.204,Z 483.927,A -85,B 0,C 180,E1 -6223.28,E2 -6223.28} C_VEL
LIN {X 0,Y 497.598,Z 471.527,A -85,B 0,C 180,E1 -6223.841,E2 -6223.841} C_VEL
LIN {X 0,Y 497.887,Z 458.76,A -85,B 0,C 180,E1 -6224.25,E2 -6224.25} C_VEL
LIN {X 0,Y 498.092,Z 445.28,A -85,B 0,C 180,E1 -6224.505,E2 -6224.505} C_VEL
LIN {X 0,Y 498.463,Z 359.319,A -85,B 0,C 180,E1 -6225.754,E2 -6225.754} C_VEL
LIN {X 0,Y 496.264,Z 345.331,A -85,B 0,C 180,E1 -6226.037,E2 -6226.037} C_VEL
LIN {X 0,Y 496.818,Z 327.581,A -85,B 0,C 180,E1 -6228.988,E2 -6228.988} C_VEL
LIN {X 0,Y 497.365,Z 309.723,A -85,B 0,C 180,E1 -6231.991,E2 -6231.991} C_VEL
LIN {X 0,Y 497.375,Z 302.047,A -85,B 0,C 180,E1 -6233.307,E2 -6233.307} C_VEL
LIN {X 0,Y 495.741,Z 293.735,A -85,B 0,C 180,E1 -6234.83,E2 -6234.83} C_VEL
LIN {X 0,Y 495.787,Z 293.726,A -85,B 0,C 180,E1 -6236.976,E2 -6236.976} C_VEL
LIN {X 0,Y 495.77,Z 293.733,A -85,B 0,C 180,E1 -6239.747,E2 -6239.747} C_VEL
LIN {X 0,Y 495.772,Z 293.724,A -85,B 0,C 180,E1 -6242.595,E2 -6242.595} C_VEL
LIN {X 0,Y 495.749,Z 293.729,A -85,B 0,C 180,E1 -6245.538,E2 -6245.538} C_VEL
LIN {X 0,Y 495.762,Z 293.726,A -85,B 0,C 180,E1 -6248.768,E2 -6248.768} C_VEL
LIN {X 0,Y 495.749,Z 293.729,A -85,B 0,C 180,E1 -6251.783,E2 -6251.783} C_VEL
LIN {X 0,Y 495.741,Z 293.728,A -85,B 0,C 180,E1 -6255.141,E2 -6255.141} C_VEL
LIN {X 0,Y 495.755,Z 293.731,A -85,B 0,C 180,E1 -6258.218,E2 -6258.218} C_VEL
LIN {X 0,Y 495.753,Z 293.726,A -85,B 0,C 180,E1 -6261.408,E2 -6261.408} C_VEL
LIN {X 0,Y 495.749,Z 293.732,A -85,B 0,C 180,E1 -6264.462,E2 -6264.462} C_VEL
LIN {X 0,Y 495.771,Z 293.726,A -85,B 0,C 180,E1 -6267.406,E2 -6267.406} C_VEL
LIN {X 0,Y 495.766,Z 293.725,A -85,B 0,C 180,E1 -6270.253,E2 -6270.253} C_VEL
LIN {X 0,Y 495.778,Z 293.73,A -85,B 0,C 180,E1 -6273.262,E2 -6273.262} C_VEL
LIN {X 0,Y 495.742,Z 293.729,A -85,B 0,C 180,E1 -6276.612,E2 -6276.612} C_VEL
LIN {X 0,Y 495.783,Z 293.732,A -85,B 0,C 180,E1 -6279.324,E2 -6279.324} C_VEL
LIN {X 0,Y 495.785,Z 293.725,A -85,B 0,C 180,E1 -6281.828,E2 -6281.828} C_VEL
LIN {X 0,Y 495.828,Z 293.716,A -85,B 0,C 180,E1 -6284.548,E2 -6284.548} C_VEL
LIN {X 0,Y 495.832,Z 293.721,A -85,B 0,C 180,E1 -6287.965,E2 -6287.965} C_VEL
LIN {X 0,Y 495.813,Z 293.719,A -85,B 0,C 180,E1 -6291.03,E2 -6291.03} C_VEL
LIN {X 0,Y 495.857,Z 293.717,A -85,B 0,C 180,E1 -6293.489,E2 -6293.489} C_VEL
LIN {X 0,Y 495.72,Z 293.74,A -85,B 0,C 180,E1 -6295.935,E2 -6295.935} C_VEL
LIN {X 0,Y 495.988,Z 293.7,A -85,B 0,C 180,E1 -6297.563,E2 -6297.563} C_VEL
LIN {X 0,Y 495.944,Z 293.703,A -85,B 0,C 180,E1 -6300.812,E2 -6300.812} C_VEL
LIN {X 0,Y 495.988,Z 293.702,A -85,B 0,C 180,E1 -6302.436,E2 -6302.436} C_VEL
LIN {X 0,Y 495.874,Z 293.712,A -85,B 0,C 180,E1 -6305.694,E2 -6305.694} C_VEL
LIN {X 0,Y 495.84,Z 293.717,A -85,B 0,C 180,E1 -6308.97,E2 -6308.97} C_VEL
LIN {X 0,Y 495.832,Z 293.718,A -85,B 0,C 180,E1 -6312.034,E2 -6312.034} C_VEL
LIN {X 0,Y 495.827,Z 293.717,A -85,B 0,C 180,E1 -6315.451,E2 -6315.451} C_VEL
LIN {X 0,Y 495.781,Z 293.724,A -85,B 0,C 180,E1 -6318.237,E2 -6318.237} C_VEL
LIN {X 0,Y 495.777,Z 293.73,A -85,B 0,C 180,E1 -6320.756,E2 -6320.756} C_VEL
LIN {X 0,Y 495.744,Z 293.731,A -85,B 0,C 180,E1 -6323.387,E2 -6323.387} C_VEL
LIN {X 0,Y 495.777,Z 293.727,A -85,B 0,C 180,E1 -6326.738,E2 -6326.738} C_VEL
LIN {X 0,Y 495.765,Z 293.727,A -85,B 0,C 180,E1 -6329.746,E2 -6329.746} C_VEL
LIN {X 0,Y 495.768,Z 293.724,A -85,B 0,C 180,E1 -6332.594,E2 -6332.594} C_VEL
LIN {X 0,Y 495.746,Z 293.736,A -85,B 0,C 180,E1 -6335.538,E2 -6335.538} C_VEL
LIN {X 0,Y 495.765,Z 293.725,A -85,B 0,C 180,E1 -6338.768,E2 -6338.768} C_VEL
LIN {X 0,Y 495.752,Z 293.735,A -85,B 0,C 180,E1 -6341.781,E2 -6341.781} C_VEL
LIN {X 0,Y 495.739,Z 293.728,A -85,B 0,C 180,E1 -6345.14,E2 -6345.14} C_VEL
LIN {X 0,Y 495.752,Z 293.731,A -85,B 0,C 180,E1 -6348.218,E2 -6348.218} C_VEL
LIN {X 0,Y 495.748,Z 293.728,A -85,B 0,C 180,E1 -6351.408,E2 -6351.408} C_VEL
LIN {X 0,Y 495.747,Z 293.732,A -85,B 0,C 180,E1 -6354.462,E2 -6354.462} C_VEL
LIN {X 0,Y 495.769,Z 293.724,A -85,B 0,C 180,E1 -6357.405,E2 -6357.405} C_VEL
LIN {X 0,Y 495.765,Z 293.731,A -85,B 0,C 180,E1 -6360.253,E2 -6360.253} C_VEL
LIN {X 0,Y 495.739,Z 293.729,A -85,B 0,C 180,E1 -6360.747,E2 -6360.747} C_VEL
LIN {X 0,Y 495.066,Z 293.814,A -85,B 0,C 180,E1 -6361.426,E2 -6361.426} C_VEL
LIN {X 0,Y 492.199,Z 294.178,A -85,B 0,C 180,E1 -6362.528,E2 -6362.528} C_VEL
LIN {X 0,Y 489.79,Z 294.473,A -85,B 0,C 180,E1 -6363.416,E2 -6363.416} C_VEL
LIN {X 0,Y 488.774,Z 294.598,A -85,B 0,C 180,E1 -6364.102,E2 -6364.102} C_VEL
LIN {X 0,Y 488.702,Z 294.61,A -85,B 0,C 180,E1 -6364.334,E2 -6364.334} C_VEL
LIN {X 0,Y 488.722,Z 294.605,A -85,B 0,C 180,E1 -6367.153,E2 -6367.153} C_VEL
LIN {X 0,Y 488.724,Z 294.601,A -85,B 0,C 180,E1 -6369.81,E2 -6369.81} C_VEL
LIN {X 0,Y 488.71,Z 294.606,A -85,B 0,C 180,E1 -6372.422,E2 -6372.422} C_VEL
LIN {X 0,Y 488.761,Z 294.607,A -85,B 0,C 180,E1 -6374.999,E2 -6374.999} C_VEL
LIN {X 0,Y 488.805,Z 294.592,A -85,B 0,C 180,E1 -6378.387,E2 -6378.387} C_VEL
LIN {X 0,Y 488.784,Z 294.602,A -85,B 0,C 180,E1 -6381.732,E2 -6381.732} C_VEL
LIN {X 0,Y 488.872,Z 294.742,A -85,B 0,C 180,E1 -6382.924,E2 -6382.924} C_VEL
LIN {X 0,Y 489.703,Z 300.139,A -85,B 0,C 180,E1 -6384.027,E2 -6384.027} C_VEL
LIN {X 0,Y 489.45,Z 312.861,A -85,B 0,C 180,E1 -6386.501,E2 -6386.501} C_VEL
LIN {X 0,Y 489.273,Z 319.574,A -85,B 0,C 180,E1 -6387.797,E2 -6387.797} C_VEL
LIN {X 0,Y 491.823,Z 333.395,A -85,B 0,C 180,E1 -6388.091,E2 -6388.091} C_VEL
LIN {X 0,Y 491.145,Z 426.988,A -85,B 0,C 180,E1 -6389.487,E2 -6389.487} C_VEL
LIN {X 0,Y 490.88,Z 439.275,A -85,B 0,C 180,E1 -6389.82,E2 -6389.82} C_VEL
LIN {X 0,Y 490.558,Z 452.556,A -85,B 0,C 180,E1 -6390.358,E2 -6390.358} C_VEL
LIN {X 0,Y 490.196,Z 464.528,A -85,B 0,C 180,E1 -6391.026,E2 -6391.026} C_VEL
LIN {X 0,Y 489.742,Z 475.95,A -85,B 0,C 180,E1 -6391.85,E2 -6391.85} C_VEL
LIN {X 0,Y 489.38,Z 486.23,A -85,B 0,C 180,E1 -6392.777,E2 -6392.777} C_VEL
LIN {X 0,Y 488.992,Z 494.682,A -85,B 0,C 180,E1 -6393.707,E2 -6393.707} C_VEL
LIN {X 0,Y 488.704,Z 502.477,A -85,B 0,C 180,E1 -6394.742,E2 -6394.742} C_VEL
LIN {X 0,Y 488.414,Z 510.085,A -85,B 0,C 180,E1 -6395.982,E2 -6395.982} C_VEL
LIN {X 0,Y 488.23,Z 517.159,A -85,B 0,C 180,E1 -6397.443,E2 -6397.443} C_VEL
LIN {X 0,Y 488.04,Z 521.87,A -85,B 0,C 180,E1 -6398.696,E2 -6398.696} C_VEL
LIN {X 0,Y 487.965,Z 525.465,A -85,B 0,C 180,E1 -6399.952,E2 -6399.952} C_VEL
LIN {X 0,Y 487.913,Z 527.31,A -85,B 0,C 180,E1 -6400.792,E2 -6400.792} C_VEL
LIN {X 0,Y 487.925,Z 528.685,A -85,B 0,C 180,E1 -6401.633,E2 -6401.633} C_VEL
LIN {X 0,Y 487.841,Z 529.666,A -85,B 0,C 180,E1 -6402.479,E2 -6402.479} C_VEL
LIN {X 0,Y 487.816,Z 530.248,A -85,B 0,C 180,E1 -6403.326,E2 -6403.326} C_VEL
LIN {X 0,Y 487.847,Z 530.383,A -85,B 0,C 180,E1 -6404.175,E2 -6404.175} C_VEL
LIN {X 0,Y 487.877,Z 530.016,A -85,B 0,C 180,E1 -6405.171,E2 -6405.171} C_VEL
LIN {X 0,Y 487.819,Z 528.291,A -85,B 0,C 180,E1 -6406.746,E2 -6406.746} C_VEL
LIN {X 0,Y 487.971,Z 525.608,A -85,B 0,C 180,E1 -6408.091,E2 -6408.091} C_VEL
LIN {X 0,Y 488.068,Z 522.09,A -85,B 0,C 180,E1 -6409.34,E2 -6409.34} C_VEL
LIN {X 0,Y 488.2,Z 517.179,A -85,B 0,C 180,E1 -6410.655,E2 -6410.655} C_VEL
LIN {X 0,Y 488.395,Z 510.893,A -85,B 0,C 180,E1 -6411.97,E2 -6411.97} C_VEL
LIN {X 0,Y 488.761,Z 502.754,A -85,B 0,C 180,E1 -6413.32,E2 -6413.32} C_VEL
LIN {X 0,Y 489.068,Z 494.635,A -85,B 0,C 180,E1 -6414.401,E2 -6414.401} C_VEL
LIN {X 0,Y 489.443,Z 484.319,A -85,B 0,C 180,E1 -6415.516,E2 -6415.516} C_VEL
LIN {X 0,Y 489.857,Z 474.086,A -85,B 0,C 180,E1 -6416.407,E2 -6416.407} C_VEL
LIN {X 0,Y 490.293,Z 462.697,A -85,B 0,C 180,E1 -6417.195,E2 -6417.195} C_VEL
LIN {X 0,Y 490.614,Z 450.145,A -85,B 0,C 180,E1 -6417.861,E2 -6417.861} C_VEL
LIN {X 0,Y 490.937,Z 436.988,A -85,B 0,C 180,E1 -6418.364,E2 -6418.364} C_VEL
LIN {X 0,Y 491.213,Z 423.639,A -85,B 0,C 180,E1 -6418.682,E2 -6418.682} C_VEL
LIN {X 0,Y 491.724,Z 331.977,A -85,B 0,C 180,E1 -6420.046,E2 -6420.046} C_VEL
LIN {X 0,Y 489.315,Z 319.386,A -85,B 0,C 180,E1 -6420.338,E2 -6420.338} C_VEL
LIN {X 0,Y 489.693,Z 303.255,A -85,B 0,C 180,E1 -6423.351,E2 -6423.351} C_VEL
LIN {X 0,Y 489.396,Z 298.291,A -85,B 0,C 180,E1 -6424.308,E2 -6424.308} C_VEL
LIN {X 0,Y 488.72,Z 294.611,A -85,B 0,C 180,E1 -6425.055,E2 -6425.055} C_VEL
LIN {X 0,Y 488.671,Z 294.614,A -85,B 0,C 180,E1 -6428.2,E2 -6428.2} C_VEL
LIN {X 0,Y 488.673,Z 294.612,A -85,B 0,C 180,E1 -6431.418,E2 -6431.418} C_VEL
LIN {X 0,Y 488.694,Z 294.613,A -85,B 0,C 180,E1 -6434.802,E2 -6434.802} C_VEL
LIN {X 0,Y 488.659,Z 294.614,A -85,B 0,C 180,E1 -6437.471,E2 -6437.471} C_VEL
LIN {X 0,Y 488.685,Z 294.61,A -85,B 0,C 180,E1 -6440.744,E2 -6440.744} C_VEL
LIN {X 0,Y 488.669,Z 294.612,A -85,B 0,C 180,E1 -6443.867,E2 -6443.867} C_VEL
LIN {X 0,Y 488.694,Z 294.6,A -85,B 0,C 180,E1 -6446.874,E2 -6446.874} C_VEL
LIN {X 0,Y 488.713,Z 294.607,A -85,B 0,C 180,E1 -6449.78,E2 -6449.78} C_VEL
LIN {X 0,Y 488.688,Z 294.609,A -85,B 0,C 180,E1 -6453.078,E2 -6453.078} C_VEL
LIN {X 0,Y 488.66,Z 294.612,A -85,B 0,C 180,E1 -6456.253,E2 -6456.253} C_VEL
LIN {X 0,Y 488.737,Z 294.601,A -85,B 0,C 180,E1 -6459.176,E2 -6459.176} C_VEL
LIN {X 0,Y 488.737,Z 294.606,A -85,B 0,C 180,E1 -6461.632,E2 -6461.632} C_VEL
LIN {X 0,Y 488.731,Z 294.601,A -85,B 0,C 180,E1 -6464.999,E2 -6464.999} C_VEL
LIN {X 0,Y 488.773,Z 294.601,A -85,B 0,C 180,E1 -6468.387,E2 -6468.387} C_VEL
LIN {X 0,Y 488.743,Z 294.598,A -85,B 0,C 180,E1 -6471.733,E2 -6471.733} C_VEL
LIN {X 0,Y 488.79,Z 294.602,A -85,B 0,C 180,E1 -6474.224,E2 -6474.224} C_VEL
LIN {X 0,Y 488.926,Z 294.574,A -85,B 0,C 180,E1 -6477.529,E2 -6477.529} C_VEL
LIN {X 0,Y 488.882,Z 294.583,A -85,B 0,C 180,E1 -6480.824,E2 -6480.824} C_VEL
LIN {X 0,Y 488.928,Z 294.579,A -85,B 0,C 180,E1 -6482.472,E2 -6482.472} C_VEL
LIN {X 0,Y 488.822,Z 294.59,A -85,B 0,C 180,E1 -6485.776,E2 -6485.776} C_VEL
LIN {X 0,Y 488.752,Z 294.596,A -85,B 0,C 180,E1 -6488.268,E2 -6488.268} C_VEL
LIN {X 0,Y 488.794,Z 294.592,A -85,B 0,C 180,E1 -6491.613,E2 -6491.613} C_VEL
LIN {X 0,Y 488.744,Z 294.606,A -85,B 0,C 180,E1 -6495.001,E2 -6495.001} C_VEL
LIN {X 0,Y 488.737,Z 294.597,A -85,B 0,C 180,E1 -6498.443,E2 -6498.443} C_VEL
LIN {X 0,Y 488.698,Z 294.613,A -85,B 0,C 180,E1 -6501.071,E2 -6501.071} C_VEL
LIN {X 0,Y 488.661,Z 294.61,A -85,B 0,C 180,E1 -6503.747,E2 -6503.747} C_VEL
LIN {X 0,Y 488.692,Z 294.61,A -85,B 0,C 180,E1 -6506.923,E2 -6506.923} C_VEL
LIN {X 0,Y 488.714,Z 294.604,A -85,B 0,C 180,E1 -6510.22,E2 -6510.22} C_VEL
LIN {X 0,Y 488.728,Z 294.611,A -85,B 0,C 180,E1 -6513.485,E2 -6513.485} C_VEL
LIN {X 0,Y 488.667,Z 294.61,A -85,B 0,C 180,E1 -6516.354,E2 -6516.354} C_VEL
LIN {X 0,Y 488.688,Z 294.609,A -85,B 0,C 180,E1 -6519.256,E2 -6519.256} C_VEL
LIN {X 0,Y 488.683,Z 294.603,A -85,B 0,C 180,E1 -6522.527,E2 -6522.527} C_VEL
LIN {X 0,Y 488.696,Z 294.607,A -85,B 0,C 180,E1 -6525.198,E2 -6525.198} C_VEL
LIN {X 0,Y 488.69,Z 294.61,A -85,B 0,C 180,E1 -6528.584,E2 -6528.584} C_VEL
LIN {X 0,Y 488.699,Z 294.608,A -85,B 0,C 180,E1 -6530.948,E2 -6530.948} C_VEL
LIN {X 0,Y 488.666,Z 294.616,A -85,B 0,C 180,E1 -6533.868,E2 -6533.868} C_VEL
LIN {X 0,Y 488.736,Z 294.604,A -85,B 0,C 180,E1 -6536.878,E2 -6536.878} C_VEL
LIN {X 0,Y 488.721,Z 294.609,A -85,B 0,C 180,E1 -6539.782,E2 -6539.782} C_VEL
LIN {X 0,Y 488.729,Z 294.61,A -85,B 0,C 180,E1 -6542.603,E2 -6542.603} C_VEL
LIN {X 0,Y 488.717,Z 294.727,A -85,B 0,C 180,E1 -6544.988,E2 -6544.988} C_VEL
LIN {X 0,Y 490.588,Z 304.996,A -85,B 0,C 180,E1 -6546.899,E2 -6546.899} C_VEL
LIN {X 0,Y 490.091,Z 319.692,A -85,B 0,C 180,E1 -6549.432,E2 -6549.432} C_VEL
LIN {X 0,Y 489.485,Z 337.509,A -85,B 0,C 180,E1 -6552.452,E2 -6552.452} C_VEL
LIN {X 0,Y 489.268,Z 345.025,A -85,B 0,C 180,E1 -6553.715,E2 -6553.715} C_VEL
LIN {X 0,Y 491.752,Z 361.305,A -85,B 0,C 180,E1 -6554.048,E2 -6554.048} C_VEL
LIN {X 0,Y 491.169,Z 453.233,A -85,B 0,C 180,E1 -6555.42,E2 -6555.42} C_VEL
LIN {X 0,Y 490.815,Z 465.734,A -85,B 0,C 180,E1 -6555.754,E2 -6555.754} C_VEL
LIN {X 0,Y 490.459,Z 478.659,A -85,B 0,C 180,E1 -6556.272,E2 -6556.272} C_VEL
LIN {X 0,Y 490.075,Z 491.21,A -85,B 0,C 180,E1 -6556.965,E2 -6556.965} C_VEL
LIN {X 0,Y 489.626,Z 502.544,A -85,B 0,C 180,E1 -6557.778,E2 -6557.778} C_VEL
LIN {X 0,Y 489.222,Z 512.995,A -85,B 0,C 180,E1 -6558.713,E2 -6558.713} C_VEL
LIN {X 0,Y 488.84,Z 521.541,A -85,B 0,C 180,E1 -6559.648,E2 -6559.648} C_VEL
LIN {X 0,Y 488.557,Z 529.429,A -85,B 0,C 180,E1 -6560.687,E2 -6560.687} C_VEL
LIN {X 0,Y 488.276,Z 537.135,A -85,B 0,C 180,E1 -6561.933,E2 -6561.933} C_VEL
LIN {X 0,Y 488.1,Z 544.241,A -85,B 0,C 180,E1 -6563.386,E2 -6563.386} C_VEL
LIN {X 0,Y 488.018,Z 548.971,A -85,B 0,C 180,E1 -6564.63,E2 -6564.63} C_VEL
LIN {X 0,Y 487.927,Z 552.586,A -85,B 0,C 180,E1 -6565.871,E2 -6565.871} C_VEL
LIN {X 0,Y 487.964,Z 554.453,A -85,B 0,C 180,E1 -6566.698,E2 -6566.698} C_VEL
LIN {X 0,Y 487.891,Z 556.85,A -85,B 0,C 180,E1 -6568.35,E2 -6568.35} C_VEL
LIN {X 0,Y 487.82,Z 557.677,A -85,B 0,C 180,E1 -6570.001,E2 -6570.001} C_VEL
LIN {X 0,Y 487.891,Z 556.858,A -85,B 0,C 180,E1 -6571.652,E2 -6571.652} C_VEL
LIN {X 0,Y 487.965,Z 554.47,A -85,B 0,C 180,E1 -6573.303,E2 -6573.303} C_VEL
LIN {X 0,Y 487.92,Z 551.532,A -85,B 0,C 180,E1 -6574.545,E2 -6574.545} C_VEL
LIN {X 0,Y 488.024,Z 547.557,A -85,B 0,C 180,E1 -6575.786,E2 -6575.786} C_VEL
LIN {X 0,Y 488.181,Z 541.441,A -85,B 0,C 180,E1 -6577.237,E2 -6577.237} C_VEL
LIN {X 0,Y 488.36,Z 534.752,A -85,B 0,C 180,E1 -6578.483,E2 -6578.483} C_VEL
LIN {X 0,Y 488.685,Z 526.454,A -85,B 0,C 180,E1 -6579.729,E2 -6579.729} C_VEL
LIN {X 0,Y 488.993,Z 517.939,A -85,B 0,C 180,E1 -6580.769,E2 -6580.769} C_VEL
LIN {X 0,Y 489.448,Z 507.418,A -85,B 0,C 180,E1 -6581.808,E2 -6581.808} C_VEL
LIN {X 0,Y 489.826,Z 495.695,A -85,B 0,C 180,E1 -6582.736,E2 -6582.736} C_VEL
LIN {X 0,Y 490.28,Z 483.625,A -85,B 0,C 180,E1 -6583.471,E2 -6583.471} C_VEL
LIN {X 0,Y 490.674,Z 471.193,A -85,B 0,C 180,E1 -6584.041,E2 -6584.041} C_VEL
LIN {X 0,Y 491.02,Z 458.355,A -85,B 0,C 180,E1 -6584.454,E2 -6584.454} C_VEL
LIN {X 0,Y 491.224,Z 444.712,A -85,B 0,C 180,E1 -6584.712,E2 -6584.712} C_VEL
LIN {X 0,Y 491.585,Z 360.077,A -85,B 0,C 180,E1 -6585.961,E2 -6585.961} C_VEL
LIN {X 0,Y 489.295,Z 345.131,A -85,B 0,C 180,E1 -6586.267,E2 -6586.267} C_VEL
LIN {X 0,Y 489.814,Z 327.317,A -85,B 0,C 180,E1 -6589.27,E2 -6589.27} C_VEL
LIN {X 0,Y 490.408,Z 310.729,A -85,B 0,C 180,E1 -6592.098,E2 -6592.098} C_VEL
LIN {X 0,Y 490.573,Z 304.712,A -85,B 0,C 180,E1 -6593.136,E2 -6593.136} C_VEL
LIN {X 0,Y 488.705,Z 294.612,A -85,B 0,C 180,E1 -6594.993,E2 -6594.993} C_VEL
LIN {X 0,Y 488.735,Z 294.609,A -85,B 0,C 180,E1 -6597.398,E2 -6597.398} C_VEL
LIN {X 0,Y 488.712,Z 294.605,A -85,B 0,C 180,E1 -6600.363,E2 -6600.363} C_VEL
LIN {X 0,Y 488.739,Z 294.603,A -85,B 0,C 180,E1 -6603.484,E2 -6603.484} C_VEL
LIN {X 0,Y 488.677,Z 294.612,A -85,B 0,C 180,E1 -6606.353,E2 -6606.353} C_VEL
LIN {X 0,Y 488.698,Z 294.605,A -85,B 0,C 180,E1 -6609.255,E2 -6609.255} C_VEL
LIN {X 0,Y 488.691,Z 294.611,A -85,B 0,C 180,E1 -6612.526,E2 -6612.526} C_VEL
LIN {X 0,Y 488.705,Z 294.604,A -85,B 0,C 180,E1 -6615.197,E2 -6615.197} C_VEL
LIN {X 0,Y 488.699,Z 294.613,A -85,B 0,C 180,E1 -6618.583,E2 -6618.583} C_VEL
LIN {X 0,Y 488.707,Z 294.608,A -85,B 0,C 180,E1 -6620.948,E2 -6620.948} C_VEL
LIN {X 0,Y 488.673,Z 294.608,A -85,B 0,C 180,E1 -6623.867,E2 -6623.867} C_VEL
LIN {X 0,Y 488.743,Z 294.608,A -85,B 0,C 180,E1 -6626.877,E2 -6626.877} C_VEL
LIN {X 0,Y 488.727,Z 294.601,A -85,B 0,C 180,E1 -6629.781,E2 -6629.781} C_VEL
LIN {X 0,Y 488.729,Z 294.611,A -85,B 0,C 180,E1 -6633.072,E2 -6633.072} C_VEL
LIN {X 0,Y 488.672,Z 294.608,A -85,B 0,C 180,E1 -6636.253,E2 -6636.253} C_VEL
LIN {X 0,Y 488.75,Z 294.606,A -85,B 0,C 180,E1 -6639.176,E2 -6639.176} C_VEL
LIN {X 0,Y 488.753,Z 294.604,A -85,B 0,C 180,E1 -6641.631,E2 -6641.631} C_VEL
LIN {X 0,Y 488.765,Z 294.599,A -85,B 0,C 180,E1 -6644.999,E2 -6644.999} C_VEL
LIN {X 0,Y 488.809,Z 294.592,A -85,B 0,C 180,E1 -6648.387,E2 -6648.387} C_VEL
LIN {X 0,Y 488.78,Z 294.603,A -85,B 0,C 180,E1 -6651.733,E2 -6651.733} C_VEL
LIN {X 0,Y 488.846,Z 294.591,A -85,B 0,C 180,E1 -6654.224,E2 -6654.224} C_VEL
LIN {X 0,Y 488.955,Z 294.575,A -85,B 0,C 180,E1 -6657.528,E2 -6657.528} C_VEL
LIN {X 0,Y 488.972,Z 294.579,A -85,B 0,C 180,E1 -6660,E2 -6660} C_VEL
LIN {X 0,Y 488.955,Z 294.578,A -85,B 0,C 180,E1 -6662.471,E2 -6662.471} C_VEL
LIN {X 0,Y 488.831,Z 294.59,A -85,B 0,C 180,E1 -6665.776,E2 -6665.776} C_VEL
LIN {X 0,Y 488.789,Z 294.6,A -85,B 0,C 180,E1 -6668.267,E2 -6668.267} C_VEL
LIN {X 0,Y 488.808,Z 294.591,A -85,B 0,C 180,E1 -6671.612,E2 -6671.612} C_VEL
LIN {X 0,Y 488.768,Z 294.601,A -85,B 0,C 180,E1 -6675,E2 -6675} C_VEL
LIN {X 0,Y 488.75,Z 294.602,A -85,B 0,C 180,E1 -6678.442,E2 -6678.442} C_VEL
LIN {X 0,Y 488.71,Z 294.61,A -85,B 0,C 180,E1 -6681.07,E2 -6681.07} C_VEL
LIN {X 0,Y 488.677,Z 294.608,A -85,B 0,C 180,E1 -6683.746,E2 -6683.746} C_VEL
LIN {X 0,Y 488.72,Z 294.603,A -85,B 0,C 180,E1 -6686.474,E2 -6686.474} C_VEL
LIN {X 0,Y 488.712,Z 294.612,A -85,B 0,C 180,E1 -6689.271,E2 -6689.271} C_VEL
LIN {X 0,Y 488.704,Z 294.604,A -85,B 0,C 180,E1 -6692.147,E2 -6692.147} C_VEL
LIN {X 0,Y 488.716,Z 294.607,A -85,B 0,C 180,E1 -6695.115,E2 -6695.115} C_VEL
LIN {X 0,Y 488.679,Z 294.608,A -85,B 0,C 180,E1 -6698.2,E2 -6698.2} C_VEL
LIN {X 0,Y 488.72,Z 294.603,A -85,B 0,C 180,E1 -6700.344,E2 -6700.344} C_VEL
LIN {X 0,Y 488.679,Z 294.615,A -85,B 0,C 180,E1 -6703.655,E2 -6703.655} C_VEL
LIN {X 0,Y 488.68,Z 294.61,A -85,B 0,C 180,E1 -6706.344,E2 -6706.344} C_VEL
LIN {X 0,Y 488.705,Z 294.608,A -85,B 0,C 180,E1 -6709.673,E2 -6709.673} C_VEL
LIN {X 0,Y 488.671,Z 294.609,A -85,B 0,C 180,E1 -6712.84,E2 -6712.84} C_VEL
LIN {X 0,Y 488.732,Z 294.605,A -85,B 0,C 180,E1 -6715.887,E2 -6715.887} C_VEL
LIN {X 0,Y 488.694,Z 294.608,A -85,B 0,C 180,E1 -6718.82,E2 -6718.82} C_VEL
LIN {X 0,Y 488.714,Z 294.603,A -85,B 0,C 180,E1 -6721.669,E2 -6721.669} C_VEL
LIN {X 0,Y 488.702,Z 294.61,A -85,B 0,C 180,E1 -6724.334,E2 -6724.334} C_VEL
LIN {X 0,Y 488.061,Z 294.696,A -85,B 0,C 180,E1 -6725.022,E2 -6725.022} C_VEL
LIN {X 0,Y 485.208,Z 295.048,A -85,B 0,C 180,E1 -6726.139,E2 -6726.139} C_VEL
LIN {X 0,Y 482.776,Z 295.347,A -85,B 0,C 180,E1 -6727.039,E2 -6727.039} C_VEL
LIN {X 0,Y 481.724,Z 295.474,A -85,B 0,C 180,E1 -6727.735,E2 -6727.735} C_VEL
LIN {X 0,Y 481.636,Z 295.485,A -85,B 0,C 180,E1 -6727.971,E2 -6727.971} C_VEL
LIN {X 0,Y 481.703,Z 295.479,A -85,B 0,C 180,E1 -6730.392,E2 -6730.392} C_VEL
LIN {X 0,Y 481.675,Z 295.487,A -85,B 0,C 180,E1 -6733.033,E2 -6733.033} C_VEL
LIN {X 0,Y 481.685,Z 295.48,A -85,B 0,C 180,E1 -6735.638,E2 -6735.638} C_VEL
LIN {X 0,Y 481.751,Z 295.47,A -85,B 0,C 180,E1 -6738.214,E2 -6738.214} C_VEL
LIN {X 0,Y 481.739,Z 295.48,A -85,B 0,C 180,E1 -6741.611,E2 -6741.611} C_VEL
LIN {X 0,Y 481.841,Z 295.475,A -85,B 0,C 180,E1 -6742.753,E2 -6742.753} C_VEL
LIN {X 0,Y 482.723,Z 301.238,A -85,B 0,C 180,E1 -6743.94,E2 -6743.94} C_VEL
LIN {X 0,Y 482.465,Z 314.002,A -85,B 0,C 180,E1 -6746.45,E2 -6746.45} C_VEL
LIN {X 0,Y 482.309,Z 319.766,A -85,B 0,C 180,E1 -6747.572,E2 -6747.572} C_VEL
LIN {X 0,Y 484.958,Z 333.601,A -85,B 0,C 180,E1 -6747.871,E2 -6747.871} C_VEL
LIN {X 0,Y 484.266,Z 426.627,A -85,B 0,C 180,E1 -6749.272,E2 -6749.272} C_VEL
LIN {X 0,Y 484.009,Z 439.097,A -85,B 0,C 180,E1 -6749.609,E2 -6749.609} C_VEL
LIN {X 0,Y 483.674,Z 452.489,A -85,B 0,C 180,E1 -6750.155,E2 -6750.155} C_VEL
LIN {X 0,Y 483.286,Z 464.556,A -85,B 0,C 180,E1 -6750.832,E2 -6750.832} C_VEL
LIN {X 0,Y 482.791,Z 476.029,A -85,B 0,C 180,E1 -6751.668,E2 -6751.668} C_VEL
LIN {X 0,Y 482.405,Z 486.333,A -85,B 0,C 180,E1 -6752.609,E2 -6752.609} C_VEL
LIN {X 0,Y 481.989,Z 494.802,A -85,B 0,C 180,E1 -6753.552,E2 -6753.552} C_VEL
LIN {X 0,Y 481.686,Z 502.609,A -85,B 0,C 180,E1 -6754.602,E2 -6754.602} C_VEL
LIN {X 0,Y 481.352,Z 510.266,A -85,B 0,C 180,E1 -6755.865,E2 -6755.865} C_VEL
LIN {X 0,Y 481.197,Z 516.231,A -85,B 0,C 180,E1 -6757.088,E2 -6757.088} C_VEL
LIN {X 0,Y 480.995,Z 521.318,A -85,B 0,C 180,E1 -6758.401,E2 -6758.401} C_VEL
LIN {X 0,Y 480.899,Z 525.101,A -85,B 0,C 180,E1 -6759.674,E2 -6759.674} C_VEL
LIN {X 0,Y 480.825,Z 527.859,A -85,B 0,C 180,E1 -6760.953,E2 -6760.953} C_VEL
LIN {X 0,Y 480.807,Z 529.157,A -85,B 0,C 180,E1 -6761.808,E2 -6761.808} C_VEL
LIN {X 0,Y 480.754,Z 530.058,A -85,B 0,C 180,E1 -6762.666,E2 -6762.666} C_VEL
LIN {X 0,Y 480.718,Z 530.506,A -85,B 0,C 180,E1 -6763.527,E2 -6763.527} C_VEL
LIN {X 0,Y 480.745,Z 530.543,A -85,B 0,C 180,E1 -6764.389,E2 -6764.389} C_VEL
LIN {X 0,Y 480.786,Z 530.179,A -85,B 0,C 180,E1 -6765.254,E2 -6765.254} C_VEL
LIN {X 0,Y 480.709,Z 529.391,A -85,B 0,C 180,E1 -6766.127,E2 -6766.127} C_VEL
LIN {X 0,Y 480.743,Z 528.131,A -85,B 0,C 180,E1 -6767,E2 -6767} C_VEL
LIN {X 0,Y 480.907,Z 525.666,A -85,B 0,C 180,E1 -6768.211,E2 -6768.211} C_VEL
LIN {X 0,Y 481.006,Z 521.573,A -85,B 0,C 180,E1 -6769.636,E2 -6769.636} C_VEL
LIN {X 0,Y 481.184,Z 516.243,A -85,B 0,C 180,E1 -6771.022,E2 -6771.022} C_VEL
LIN {X 0,Y 481.43,Z 509.961,A -85,B 0,C 180,E1 -6772.305,E2 -6772.305} C_VEL
LIN {X 0,Y 481.744,Z 503.196,A -85,B 0,C 180,E1 -6773.424,E2 -6773.424} C_VEL
LIN {X 0,Y 482.07,Z 494.907,A -85,B 0,C 180,E1 -6774.55,E2 -6774.55} C_VEL
LIN {X 0,Y 482.449,Z 485.368,A -85,B 0,C 180,E1 -6775.606,E2 -6775.606} C_VEL
LIN {X 0,Y 482.916,Z 474.433,A -85,B 0,C 180,E1 -6776.583,E2 -6776.583} C_VEL
LIN {X 0,Y 483.419,Z 462.694,A -85,B 0,C 180,E1 -6777.407,E2 -6777.407} C_VEL
LIN {X 0,Y 483.742,Z 450.674,A -85,B 0,C 180,E1 -6778.056,E2 -6778.056} C_VEL
LIN {X 0,Y 484.091,Z 437.716,A -85,B 0,C 180,E1 -6778.566,E2 -6778.566} C_VEL
LIN {X 0,Y 484.365,Z 425.611,A -85,B 0,C 180,E1 -6778.874,E2 -6778.874} C_VEL
LIN {X 0,Y 484.961,Z 333.004,A -85,B 0,C 180,E1 -6780.275,E2 -6780.275} C_VEL
LIN {X 0,Y 482.377,Z 319.519,A -85,B 0,C 180,E1 -6780.599,E2 -6780.599} C_VEL
LIN {X 0,Y 482.768,Z 303.746,A -85,B 0,C 180,E1 -6783.585,E2 -6783.585} C_VEL
LIN {X 0,Y 482.257,Z 298.41,A -85,B 0,C 180,E1 -6784.634,E2 -6784.634} C_VEL
LIN {X 0,Y 481.676,Z 295.488,A -85,B 0,C 180,E1 -6785.242,E2 -6785.242} C_VEL
LIN {X 0,Y 481.66,Z 295.491,A -85,B 0,C 180,E1 -6788.859,E2 -6788.859} C_VEL
LIN {X 0,Y 481.633,Z 295.487,A -85,B 0,C 180,E1 -6792.161,E2 -6792.161} C_VEL
LIN {X 0,Y 481.646,Z 295.488,A -85,B 0,C 180,E1 -6795.541,E2 -6795.541} C_VEL
LIN {X 0,Y 481.618,Z 295.493,A -85,B 0,C 180,E1 -6798.954,E2 -6798.954} C_VEL
LIN {X 0,Y 481.644,Z 295.485,A -85,B 0,C 180,E1 -6801.993,E2 -6801.993} C_VEL
LIN {X 0,Y 481.675,Z 295.481,A -85,B 0,C 180,E1 -6805.317,E2 -6805.317} C_VEL
LIN {X 0,Y 481.633,Z 295.487,A -85,B 0,C 180,E1 -6808.311,E2 -6808.311} C_VEL
LIN {X 0,Y 481.663,Z 295.484,A -85,B 0,C 180,E1 -6811.216,E2 -6811.216} C_VEL
LIN {X 0,Y 481.617,Z 295.49,A -85,B 0,C 180,E1 -6814.038,E2 -6814.038} C_VEL
LIN {X 0,Y 481.665,Z 295.482,A -85,B 0,C 180,E1 -6816.812,E2 -6816.812} C_VEL
LIN {X 0,Y 481.685,Z 295.483,A -85,B 0,C 180,E1 -6819.502,E2 -6819.502} C_VEL
LIN {X 0,Y 481.659,Z 295.486,A -85,B 0,C 180,E1 -6822.157,E2 -6822.157} C_VEL
LIN {X 0,Y 481.711,Z 295.476,A -85,B 0,C 180,E1 -6824.775,E2 -6824.775} C_VEL
LIN {X 0,Y 481.725,Z 295.481,A -85,B 0,C 180,E1 -6828.215,E2 -6828.215} C_VEL
LIN {X 0,Y 481.701,Z 295.474,A -85,B 0,C 180,E1 -6831.611,E2 -6831.611} C_VEL
LIN {X 0,Y 481.752,Z 295.477,A -85,B 0,C 180,E1 -6834.139,E2 -6834.139} C_VEL
LIN {X 0,Y 481.892,Z 295.449,A -85,B 0,C 180,E1 -6837.493,E2 -6837.493} C_VEL
LIN {X 0,Y 481.835,Z 295.461,A -85,B 0,C 180,E1 -6840.836,E2 -6840.836} C_VEL
LIN {X 0,Y 481.894,Z 295.455,A -85,B 0,C 180,E1 -6842.508,E2 -6842.508} C_VEL
LIN {X 0,Y 481.783,Z 295.467,A -85,B 0,C 180,E1 -6845.861,E2 -6845.861} C_VEL
LIN {X 0,Y 481.709,Z 295.474,A -85,B 0,C 180,E1 -6848.389,E2 -6848.389} C_VEL
LIN {X 0,Y 481.74,Z 295.47,A -85,B 0,C 180,E1 -6851.785,E2 -6851.785} C_VEL
LIN {X 0,Y 481.728,Z 295.477,A -85,B 0,C 180,E1 -6855.225,E2 -6855.225} C_VEL
LIN {X 0,Y 481.699,Z 295.476,A -85,B 0,C 180,E1 -6858.722,E2 -6858.722} C_VEL
LIN {X 0,Y 481.636,Z 295.487,A -85,B 0,C 180,E1 -6861.395,E2 -6861.395} C_VEL
LIN {X 0,Y 481.64,Z 295.483,A -85,B 0,C 180,E1 -6864.115,E2 -6864.115} C_VEL
LIN {X 0,Y 481.667,Z 295.486,A -85,B 0,C 180,E1 -6867.123,E2 -6867.123} C_VEL
LIN {X 0,Y 481.664,Z 295.485,A -85,B 0,C 180,E1 -6869.742,E2 -6869.742} C_VEL
LIN {X 0,Y 481.665,Z 295.481,A -85,B 0,C 180,E1 -6872.675,E2 -6872.675} C_VEL
LIN {X 0,Y 481.625,Z 295.492,A -85,B 0,C 180,E1 -6875.711,E2 -6875.711} C_VEL
LIN {X 0,Y 481.66,Z 295.481,A -85,B 0,C 180,E1 -6878.86,E2 -6878.86} C_VEL
LIN {X 0,Y 481.635,Z 295.484,A -85,B 0,C 180,E1 -6882.162,E2 -6882.162} C_VEL
LIN {X 0,Y 481.649,Z 295.488,A -85,B 0,C 180,E1 -6885.543,E2 -6885.543} C_VEL
LIN {X 0,Y 481.645,Z 295.487,A -85,B 0,C 180,E1 -6888.958,E2 -6888.958} C_VEL
LIN {X 0,Y 481.646,Z 295.492,A -85,B 0,C 180,E1 -6891.994,E2 -6891.994} C_VEL
LIN {X 0,Y 481.685,Z 295.479,A -85,B 0,C 180,E1 -6895.319,E2 -6895.319} C_VEL
LIN {X 0,Y 481.642,Z 295.491,A -85,B 0,C 180,E1 -6898.313,E2 -6898.313} C_VEL
LIN {X 0,Y 481.696,Z 295.481,A -85,B 0,C 180,E1 -6901.219,E2 -6901.219} C_VEL
LIN {X 0,Y 481.671,Z 295.492,A -85,B 0,C 180,E1 -6904.042,E2 -6904.042} C_VEL
LIN {X 0,Y 481.679,Z 295.627,A -85,B 0,C 180,E1 -6904.773,E2 -6904.773} C_VEL
LIN {X 0,Y 483.591,Z 305.788,A -85,B 0,C 180,E1 -6906.703,E2 -6906.703} C_VEL
LIN {X 0,Y 483.364,Z 316.112,A -85,B 0,C 180,E1 -6908.52,E2 -6908.52} C_VEL
LIN {X 0,Y 482.595,Z 336.107,A -85,B 0,C 180,E1 -6911.974,E2 -6911.974} C_VEL
LIN {X 0,Y 482.286,Z 344.748,A -85,B 0,C 180,E1 -6913.449,E2 -6913.449} C_VEL
LIN {X 0,Y 484.963,Z 361.861,A -85,B 0,C 180,E1 -6913.819,E2 -6913.819} C_VEL
LIN {X 0,Y 484.323,Z 453.404,A -85,B 0,C 180,E1 -6915.209,E2 -6915.209} C_VEL
LIN {X 0,Y 483.959,Z 465.763,A -85,B 0,C 180,E1 -6915.547,E2 -6915.547} C_VEL
LIN {X 0,Y 483.55,Z 478.606,A -85,B 0,C 180,E1 -6916.072,E2 -6916.072} C_VEL
LIN {X 0,Y 483.148,Z 491.138,A -85,B 0,C 180,E1 -6916.778,E2 -6916.778} C_VEL
LIN {X 0,Y 482.669,Z 502.391,A -85,B 0,C 180,E1 -6917.599,E2 -6917.599} C_VEL
LIN {X 0,Y 482.226,Z 512.829,A -85,B 0,C 180,E1 -6918.547,E2 -6918.547} C_VEL
LIN {X 0,Y 481.835,Z 521.369,A -85,B 0,C 180,E1 -6919.496,E2 -6919.496} C_VEL
LIN {X 0,Y 481.523,Z 529.253,A -85,B 0,C 180,E1 -6920.55,E2 -6920.55} C_VEL
LIN {X 0,Y 481.226,Z 536.953,A -85,B 0,C 180,E1 -6921.815,E2 -6921.815} C_VEL
LIN {X 0,Y 481.019,Z 544.056,A -85,B 0,C 180,E1 -6923.288,E2 -6923.288} C_VEL
LIN {X 0,Y 480.93,Z 548.783,A -85,B 0,C 180,E1 -6924.55,E2 -6924.55} C_VEL
LIN {X 0,Y 480.827,Z 552.393,A -85,B 0,C 180,E1 -6925.81,E2 -6925.81} C_VEL
LIN {X 0,Y 480.888,Z 554.259,A -85,B 0,C 180,E1 -6926.649,E2 -6926.649} C_VEL
LIN {X 0,Y 480.792,Z 556.653,A -85,B 0,C 180,E1 -6928.325,E2 -6928.325} C_VEL
LIN {X 0,Y 480.76,Z 557.262,A -85,B 0,C 180,E1 -6929.163,E2 -6929.163} C_VEL
LIN {X 0,Y 480.743,Z 557.479,A -85,B 0,C 180,E1 -6930.001,E2 -6930.001} C_VEL
LIN {X 0,Y 480.792,Z 556.657,A -85,B 0,C 180,E1 -6931.676,E2 -6931.676} C_VEL
LIN {X 0,Y 480.823,Z 555.663,A -85,B 0,C 180,E1 -6932.514,E2 -6932.514} C_VEL
LIN {X 0,Y 480.888,Z 554.266,A -85,B 0,C 180,E1 -6933.352,E2 -6933.352} C_VEL
LIN {X 0,Y 480.839,Z 551.324,A -85,B 0,C 180,E1 -6934.612,E2 -6934.612} C_VEL
LIN {X 0,Y 480.928,Z 547.344,A -85,B 0,C 180,E1 -6935.872,E2 -6935.872} C_VEL
LIN {X 0,Y 481.106,Z 541.218,A -85,B 0,C 180,E1 -6937.344,E2 -6937.344} C_VEL
LIN {X 0,Y 481.319,Z 534.524,A -85,B 0,C 180,E1 -6938.608,E2 -6938.608} C_VEL
LIN {X 0,Y 481.63,Z 526.217,A -85,B 0,C 180,E1 -6939.873,E2 -6939.873} C_VEL
LIN {X 0,Y 481.983,Z 517.692,A -85,B 0,C 180,E1 -6940.928,E2 -6940.928} C_VEL
LIN {X 0,Y 482.468,Z 507.174,A -85,B 0,C 180,E1 -6941.98,E2 -6941.98} C_VEL
LIN {X 0,Y 482.873,Z 495.8,A -85,B 0,C 180,E1 -6942.894,E2 -6942.894} C_VEL
LIN {X 0,Y 483.306,Z 485.284,A -85,B 0,C 180,E1 -6943.562,E2 -6943.562} C_VEL
LIN {X 0,Y 483.757,Z 473.467,A -85,B 0,C 180,E1 -6944.138,E2 -6944.138} C_VEL
LIN {X 0,Y 484.036,Z 461.642,A -85,B 0,C 180,E1 -6944.559,E2 -6944.559} C_VEL
LIN {X 0,Y 484.297,Z 449.094,A -85,B 0,C 180,E1 -6944.847,E2 -6944.847} C_VEL
LIN {X 0,Y 484.734,Z 360.808,A -85,B 0,C 180,E1 -6946.169,E2 -6946.169} C_VEL
LIN {X 0,Y 482.306,Z 344.874,A -85,B 0,C 180,E1 -6946.509,E2 -6946.509} C_VEL
LIN {X 0,Y 482.889,Z 327.05,A -85,B 0,C 180,E1 -6949.558,E2 -6949.558} C_VEL
LIN {X 0,Y 483.516,Z 310.426,A -85,B 0,C 180,E1 -6952.43,E2 -6952.43} C_VEL
LIN {X 0,Y 483.52,Z 305.129,A -85,B 0,C 180,E1 -6953.362,E2 -6953.362} C_VEL
LIN {X 0,Y 481.658,Z 295.49,A -85,B 0,C 180,E1 -6955.182,E2 -6955.182} C_VEL
LIN {X 0,Y 481.696,Z 295.487,A -85,B 0,C 180,E1 -6957.833,E2 -6957.833} C_VEL
LIN {X 0,Y 481.648,Z 295.483,A -85,B 0,C 180,E1 -6960.711,E2 -6960.711} C_VEL
LIN {X 0,Y 481.702,Z 295.482,A -85,B 0,C 180,E1 -6963.733,E2 -6963.733} C_VEL
LIN {X 0,Y 481.624,Z 295.487,A -85,B 0,C 180,E1 -6966.748,E2 -6966.748} C_VEL
LIN {X 0,Y 481.661,Z 295.487,A -85,B 0,C 180,E1 -6969.943,E2 -6969.943} C_VEL
LIN {X 0,Y 481.63,Z 295.485,A -85,B 0,C 180,E1 -6973.146,E2 -6973.146} C_VEL
LIN {X 0,Y 481.657,Z 295.482,A -85,B 0,C 180,E1 -6975.642,E2 -6975.642} C_VEL
LIN {X 0,Y 481.653,Z 295.486,A -85,B 0,C 180,E1 -6978.958,E2 -6978.958} C_VEL
LIN {X 0,Y 481.654,Z 295.483,A -85,B 0,C 180,E1 -6981.994,E2 -6981.994} C_VEL
LIN {X 0,Y 481.691,Z 295.48,A -85,B 0,C 180,E1 -6985.318,E2 -6985.318} C_VEL
LIN {X 0,Y 481.648,Z 295.485,A -85,B 0,C 180,E1 -6988.312,E2 -6988.312} C_VEL
LIN {X 0,Y 481.679,Z 295.485,A -85,B 0,C 180,E1 -6991.217,E2 -6991.217} C_VEL
LIN {X 0,Y 481.667,Z 295.481,A -85,B 0,C 180,E1 -6994.041,E2 -6994.041} C_VEL
LIN {X 0,Y 481.678,Z 295.483,A -85,B 0,C 180,E1 -6996.812,E2 -6996.812} C_VEL
LIN {X 0,Y 481.699,Z 295.483,A -85,B 0,C 180,E1 -6999.503,E2 -6999.503} C_VEL
LIN {X 0,Y 481.695,Z 295.478,A -85,B 0,C 180,E1 -7002.158,E2 -7002.158} C_VEL
LIN {X 0,Y 481.746,Z 295.471,A -85,B 0,C 180,E1 -7004.776,E2 -7004.776} C_VEL
LIN {X 0,Y 481.754,Z 295.472,A -85,B 0,C 180,E1 -7008.215,E2 -7008.215} C_VEL
LIN {X 0,Y 481.735,Z 295.479,A -85,B 0,C 180,E1 -7011.611,E2 -7011.611} C_VEL
LIN {X 0,Y 481.806,Z 295.469,A -85,B 0,C 180,E1 -7014.139,E2 -7014.139} C_VEL
LIN {X 0,Y 481.921,Z 295.451,A -85,B 0,C 180,E1 -7017.492,E2 -7017.492} C_VEL
LIN {X 0,Y 481.943,Z 295.454,A -85,B 0,C 180,E1 -7020,E2 -7020} C_VEL
LIN {X 0,Y 481.922,Z 295.454,A -85,B 0,C 180,E1 -7022.507,E2 -7022.507} C_VEL
LIN {X 0,Y 481.791,Z 295.468,A -85,B 0,C 180,E1 -7025.861,E2 -7025.861} C_VEL
LIN {X 0,Y 481.743,Z 295.48,A -85,B 0,C 180,E1 -7028.388,E2 -7028.388} C_VEL
LIN {X 0,Y 481.754,Z 295.47,A -85,B 0,C 180,E1 -7031.785,E2 -7031.785} C_VEL
LIN {X 0,Y 481.747,Z 295.473,A -85,B 0,C 180,E1 -7035.224,E2 -7035.224} C_VEL
LIN {X 0,Y 481.711,Z 295.483,A -85,B 0,C 180,E1 -7038.722,E2 -7038.722} C_VEL
LIN {X 0,Y 481.648,Z 295.486,A -85,B 0,C 180,E1 -7041.394,E2 -7041.394} C_VEL
LIN {X 0,Y 481.658,Z 295.482,A -85,B 0,C 180,E1 -7044.114,E2 -7044.114} C_VEL
LIN {X 0,Y 481.697,Z 295.486,A -85,B 0,C 180,E1 -7047.127,E2 -7047.127} C_VEL
LIN {X 0,Y 481.674,Z 295.482,A -85,B 0,C 180,E1 -7049.741,E2 -7049.741} C_VEL
LIN {X 0,Y 481.672,Z 295.481,A -85,B 0,C 180,E1 -7052.674,E2 -7052.674} C_VEL
LIN {X 0,Y 481.633,Z 295.491,A -85,B 0,C 180,E1 -7055.71,E2 -7055.71} C_VEL
LIN {X 0,Y 481.672,Z 295.481,A -85,B 0,C 180,E1 -7058.859,E2 -7058.859} C_VEL
LIN {X 0,Y 481.648,Z 295.489,A -85,B 0,C 180,E1 -7061.912,E2 -7061.912} C_VEL
LIN {X 0,Y 481.656,Z 295.483,A -85,B 0,C 180,E1 -7064.458,E2 -7064.458} C_VEL
LIN {X 0,Y 481.645,Z 295.491,A -85,B 0,C 180,E1 -7067.838,E2 -7067.838} C_VEL
LIN {X 0,Y 481.658,Z 295.483,A -85,B 0,C 180,E1 -7070.654,E2 -7070.654} C_VEL
LIN {X 0,Y 481.623,Z 295.487,A -85,B 0,C 180,E1 -7073.377,E2 -7073.377} C_VEL
LIN {X 0,Y 481.712,Z 295.484,A -85,B 0,C 180,E1 -7076.33,E2 -7076.33} C_VEL
LIN {X 0,Y 481.652,Z 295.482,A -85,B 0,C 180,E1 -7079.417,E2 -7079.417} C_VEL
LIN {X 0,Y 481.67,Z 295.485,A -85,B 0,C 180,E1 -7082.166,E2 -7082.166} C_VEL
LIN {X 0,Y 481.676,Z 295.483,A -85,B 0,C 180,E1 -7084.967,E2 -7084.967} C_VEL
LIN {X 0,Y 481.636,Z 295.485,A -85,B 0,C 180,E1 -7087.971,E2 -7087.971} C_VEL
LIN {X 0,Y 480.969,Z 295.576,A -85,B 0,C 180,E1 -7088.669,E2 -7088.669} C_VEL
LIN {X 0,Y 478.144,Z 295.925,A -85,B 0,C 180,E1 -7089.803,E2 -7089.803} C_VEL
LIN {X 0,Y 475.758,Z 296.225,A -85,B 0,C 180,E1 -7090.717,E2 -7090.717} C_VEL
LIN {X 0,Y 474.731,Z 296.347,A -85,B 0,C 180,E1 -7091.423,E2 -7091.423} C_VEL
LIN {X 0,Y 474.646,Z 296.356,A -85,B 0,C 180,E1 -7091.662,E2 -7091.662} C_VEL
LIN {X 0,Y 474.7,Z 296.352,A -85,B 0,C 180,E1 -7094.544,E2 -7094.544} C_VEL
LIN {X 0,Y 474.704,Z 296.348,A -85,B 0,C 180,E1 -7098.037,E2 -7098.037} C_VEL
LIN {X 0,Y 474.71,Z 296.356,A -85,B 0,C 180,E1 -7101.485,E2 -7101.485} C_VEL
LIN {X 0,Y 474.796,Z 296.486,A -85,B 0,C 180,E1 -7102.631,E2 -7102.631} C_VEL
LIN {X 0,Y 475.743,Z 302.324,A -85,B 0,C 180,E1 -7103.851,E2 -7103.851} C_VEL
LIN {X 0,Y 475.48,Z 315.146,A -85,B 0,C 180,E1 -7106.398,E2 -7106.398} C_VEL
LIN {X 0,Y 475.342,Z 319.868,A -85,B 0,C 180,E1 -7107.325,E2 -7107.325} C_VEL
LIN {X 0,Y 478.119,Z 334.386,A -85,B 0,C 180,E1 -7107.656,E2 -7107.656} C_VEL
LIN {X 0,Y 477.374,Z 427.195,A -85,B 0,C 180,E1 -7109.077,E2 -7109.077} C_VEL
LIN {X 0,Y 477.119,Z 440.264,A -85,B 0,C 180,E1 -7109.445,E2 -7109.445} C_VEL
LIN {X 0,Y 476.764,Z 453.405,A -85,B 0,C 180,E1 -7109.999,E2 -7109.999} C_VEL
LIN {X 0,Y 476.372,Z 464.483,A -85,B 0,C 180,E1 -7110.633,E2 -7110.633} C_VEL
LIN {X 0,Y 475.846,Z 476.008,A -85,B 0,C 180,E1 -7111.48,E2 -7111.48} C_VEL
LIN {X 0,Y 475.43,Z 486.362,A -85,B 0,C 180,E1 -7112.435,E2 -7112.435} C_VEL
LIN {X 0,Y 474.98,Z 494.872,A -85,B 0,C 180,E1 -7113.392,E2 -7113.392} C_VEL
LIN {X 0,Y 474.657,Z 502.709,A -85,B 0,C 180,E1 -7114.458,E2 -7114.458} C_VEL
LIN {X 0,Y 474.294,Z 510.398,A -85,B 0,C 180,E1 -7115.74,E2 -7115.74} C_VEL
LIN {X 0,Y 474.176,Z 515.647,A -85,B 0,C 180,E1 -7116.809,E2 -7116.809} C_VEL
LIN {X 0,Y 473.976,Z 520.76,A -85,B 0,C 180,E1 -7118.097,E2 -7118.097} C_VEL
LIN {X 0,Y 473.814,Z 524.738,A -85,B 0,C 180,E1 -7119.39,E2 -7119.39} C_VEL
LIN {X 0,Y 473.779,Z 526.781,A -85,B 0,C 180,E1 -7120.253,E2 -7120.253} C_VEL
LIN {X 0,Y 473.729,Z 529.282,A -85,B 0,C 180,E1 -7121.724,E2 -7121.724} C_VEL
LIN {X 0,Y 473.657,Z 530.387,A -85,B 0,C 180,E1 -7122.859,E2 -7122.859} C_VEL
LIN {X 0,Y 473.619,Z 530.745,A -85,B 0,C 180,E1 -7123.734,E2 -7123.734} C_VEL
LIN {X 0,Y 473.705,Z 530.341,A -85,B 0,C 180,E1 -7125.344,E2 -7125.344} C_VEL
LIN {X 0,Y 473.628,Z 529.314,A -85,B 0,C 180,E1 -7126.375,E2 -7126.375} C_VEL
LIN {X 0,Y 473.695,Z 527.972,A -85,B 0,C 180,E1 -7127.26,E2 -7127.26} C_VEL
LIN {X 0,Y 473.83,Z 525.744,A -85,B 0,C 180,E1 -7128.329,E2 -7128.329} C_VEL
LIN {X 0,Y 473.959,Z 521.067,A -85,B 0,C 180,E1 -7129.94,E2 -7129.94} C_VEL
LIN {X 0,Y 474.146,Z 515.759,A -85,B 0,C 180,E1 -7131.298,E2 -7131.298} C_VEL
LIN {X 0,Y 474.454,Z 508.98,A -85,B 0,C 180,E1 -7132.651,E2 -7132.651} C_VEL
LIN {X 0,Y 474.837,Z 500.378,A -85,B 0,C 180,E1 -7134.017,E2 -7134.017} C_VEL
LIN {X 0,Y 475.263,Z 491.444,A -85,B 0,C 180,E1 -7135.159,E2 -7135.159} C_VEL
LIN {X 0,Y 475.703,Z 481.27,A -85,B 0,C 180,E1 -7136.206,E2 -7136.206} C_VEL
LIN {X 0,Y 476.223,Z 470.392,A -85,B 0,C 180,E1 -7137.105,E2 -7137.105} C_VEL
LIN {X 0,Y 476.695,Z 459.12,A -85,B 0,C 180,E1 -7137.844,E2 -7137.844} C_VEL
LIN {X 0,Y 477.039,Z 447.512,A -85,B 0,C 180,E1 -7138.426,E2 -7138.426} C_VEL
LIN {X 0,Y 477.341,Z 434.663,A -85,B 0,C 180,E1 -7138.887,E2 -7138.887} C_VEL
LIN {X 0,Y 477.576,Z 421.316,A -85,B 0,C 180,E1 -7139.184,E2 -7139.184} C_VEL
LIN {X 0,Y 478.225,Z 333.956,A -85,B 0,C 180,E1 -7140.514,E2 -7140.514} C_VEL
LIN {X 0,Y 475.429,Z 319.717,A -85,B 0,C 180,E1 -7140.866,E2 -7140.866} C_VEL
LIN {X 0,Y 475.817,Z 305.255,A -85,B 0,C 180,E1 -7143.633,E2 -7143.633} C_VEL
LIN {X 0,Y 475.341,Z 299.907,A -85,B 0,C 180,E1 -7144.695,E2 -7144.695} C_VEL
LIN {X 0,Y 474.613,Z 296.367,A -85,B 0,C 180,E1 -7145.469,E2 -7145.469} C_VEL
LIN {X 0,Y 474.603,Z 296.368,A -85,B 0,C 180,E1 -7148.457,E2 -7148.457} C_VEL
LIN {X 0,Y 474.602,Z 296.363,A -85,B 0,C 180,E1 -7151.786,E2 -7151.786} C_VEL
LIN {X 0,Y 474.609,Z 296.367,A -85,B 0,C 180,E1 -7154.702,E2 -7154.702} C_VEL
LIN {X 0,Y 474.576,Z 296.366,A -85,B 0,C 180,E1 -7157.768,E2 -7157.768} C_VEL
LIN {X 0,Y 474.613,Z 296.361,A -85,B 0,C 180,E1 -7160.451,E2 -7160.451} C_VEL
LIN {X 0,Y 474.58,Z 296.369,A -85,B 0,C 180,E1 -7163.676,E2 -7163.676} C_VEL
LIN {X 0,Y 474.606,Z 296.354,A -85,B 0,C 180,E1 -7166.777,E2 -7166.777} C_VEL
LIN {X 0,Y 474.592,Z 296.366,A -85,B 0,C 180,E1 -7169.769,E2 -7169.769} C_VEL
LIN {X 0,Y 474.628,Z 296.359,A -85,B 0,C 180,E1 -7172.676,E2 -7172.676} C_VEL
LIN {X 0,Y 474.615,Z 296.365,A -85,B 0,C 180,E1 -7175.505,E2 -7175.505} C_VEL
LIN {X 0,Y 474.625,Z 296.358,A -85,B 0,C 180,E1 -7178.884,E2 -7178.884} C_VEL
LIN {X 0,Y 474.623,Z 296.362,A -85,B 0,C 180,E1 -7181.883,E2 -7181.883} C_VEL
LIN {X 0,Y 474.67,Z 296.354,A -85,B 0,C 180,E1 -7184.544,E2 -7184.544} C_VEL
LIN {X 0,Y 474.683,Z 296.356,A -85,B 0,C 180,E1 -7188.037,E2 -7188.037} C_VEL
LIN {X 0,Y 474.65,Z 296.351,A -85,B 0,C 180,E1 -7191.485,E2 -7191.485} C_VEL
LIN {X 0,Y 474.716,Z 296.352,A -85,B 0,C 180,E1 -7194.052,E2 -7194.052} C_VEL
LIN {X 0,Y 474.833,Z 296.329,A -85,B 0,C 180,E1 -7197.455,E2 -7197.455} C_VEL
LIN {X 0,Y 474.865,Z 296.332,A -85,B 0,C 180,E1 -7200,E2 -7200} C_VEL
LIN {X 0,Y 474.859,Z 296.331,A -85,B 0,C 180,E1 -7202.545,E2 -7202.545} C_VEL
LIN {X 0,Y 474.746,Z 296.344,A -85,B 0,C 180,E1 -7205.948,E2 -7205.948} C_VEL
LIN {X 0,Y 474.684,Z 296.35,A -85,B 0,C 180,E1 -7208.515,E2 -7208.515} C_VEL
LIN {X 0,Y 474.694,Z 296.348,A -85,B 0,C 180,E1 -7211.963,E2 -7211.963} C_VEL
LIN {X 0,Y 474.671,Z 296.352,A -85,B 0,C 180,E1 -7215.767,E2 -7215.767} C_VEL
LIN {X 0,Y 474.653,Z 296.357,A -85,B 0,C 180,E1 -7219.011,E2 -7219.011} C_VEL
LIN {X 0,Y 474.579,Z 296.363,A -85,B 0,C 180,E1 -7221.73,E2 -7221.73} C_VEL
LIN {X 0,Y 474.618,Z 296.359,A -85,B 0,C 180,E1 -7224.495,E2 -7224.495} C_VEL
LIN {X 0,Y 474.629,Z 296.361,A -85,B 0,C 180,E1 -7227.325,E2 -7227.325} C_VEL
LIN {X 0,Y 474.594,Z 296.363,A -85,B 0,C 180,E1 -7230.231,E2 -7230.231} C_VEL
LIN {X 0,Y 474.628,Z 296.363,A -85,B 0,C 180,E1 -7233.222,E2 -7233.222} C_VEL
LIN {X 0,Y 474.578,Z 296.365,A -85,B 0,C 180,E1 -7236.325,E2 -7236.325} C_VEL
LIN {X 0,Y 474.616,Z 296.365,A -85,B 0,C 180,E1 -7239.549,E2 -7239.549} C_VEL
LIN {X 0,Y 474.592,Z 296.36,A -85,B 0,C 180,E1 -7242.234,E2 -7242.234} C_VEL
LIN {X 0,Y 474.611,Z 296.362,A -85,B 0,C 180,E1 -7245.299,E2 -7245.299} C_VEL
LIN {X 0,Y 474.611,Z 296.368,A -85,B 0,C 180,E1 -7248.215,E2 -7248.215} C_VEL
LIN {X 0,Y 474.606,Z 296.367,A -85,B 0,C 180,E1 -7251.543,E2 -7251.543} C_VEL
LIN {X 0,Y 474.619,Z 296.36,A -85,B 0,C 180,E1 -7254.726,E2 -7254.726} C_VEL
LIN {X 0,Y 474.633,Z 296.363,A -85,B 0,C 180,E1 -7257.789,E2 -7257.789} C_VEL
LIN {X 0,Y 474.62,Z 296.365,A -85,B 0,C 180,E1 -7260.886,E2 -7260.886} C_VEL
LIN {X 0,Y 474.626,Z 296.365,A -85,B 0,C 180,E1 -7263.627,E2 -7263.627} C_VEL
LIN {X 0,Y 474.644,Z 296.497,A -85,B 0,C 180,E1 -7264.542,E2 -7264.542} C_VEL
LIN {X 0,Y 476.63,Z 306.818,A -85,B 0,C 180,E1 -7266.54,E2 -7266.54} C_VEL
LIN {X 0,Y 476.522,Z 314.679,A -85,B 0,C 180,E1 -7267.955,E2 -7267.955} C_VEL
LIN {X 0,Y 475.768,Z 333.475,A -85,B 0,C 180,E1 -7271.26,E2 -7271.26} C_VEL
LIN {X 0,Y 475.337,Z 344.583,A -85,B 0,C 180,E1 -7273.19,E2 -7273.19} C_VEL
LIN {X 0,Y 478.15,Z 362.598,A -85,B 0,C 180,E1 -7273.582,E2 -7273.582} C_VEL
LIN {X 0,Y 477.51,Z 452.589,A -85,B 0,C 180,E1 -7274.966,E2 -7274.966} C_VEL
LIN {X 0,Y 477.114,Z 465.154,A -85,B 0,C 180,E1 -7275.308,E2 -7275.308} C_VEL
LIN {X 0,Y 476.681,Z 478.665,A -85,B 0,C 180,E1 -7275.867,E2 -7275.867} C_VEL
LIN {X 0,Y 476.242,Z 490.805,A -85,B 0,C 180,E1 -7276.561,E2 -7276.561} C_VEL
LIN {X 0,Y 475.726,Z 501.493,A -85,B 0,C 180,E1 -7277.344,E2 -7277.344} C_VEL
LIN {X 0,Y 475.225,Z 512.738,A -85,B 0,C 180,E1 -7278.376,E2 -7278.376} C_VEL
LIN {X 0,Y 474.824,Z 521.247,A -85,B 0,C 180,E1 -7279.339,E2 -7279.339} C_VEL
LIN {X 0,Y 474.416,Z 530.479,A -85,B 0,C 180,E1 -7280.622,E2 -7280.622} C_VEL
LIN {X 0,Y 474.114,Z 537.905,A -85,B 0,C 180,E1 -7281.905,E2 -7281.905} C_VEL
LIN {X 0,Y 473.936,Z 543.873,A -85,B 0,C 180,E1 -7283.188,E2 -7283.188} C_VEL
LIN {X 0,Y 473.845,Z 548.595,A -85,B 0,C 180,E1 -7284.469,E2 -7284.469} C_VEL
LIN {X 0,Y 473.734,Z 552.204,A -85,B 0,C 180,E1 -7285.747,E2 -7285.747} C_VEL
LIN {X 0,Y 473.795,Z 554.067,A -85,B 0,C 180,E1 -7286.599,E2 -7286.599} C_VEL
LIN {X 0,Y 473.741,Z 555.462,A -85,B 0,C 180,E1 -7287.45,E2 -7287.45} C_VEL
LIN {X 0,Y 473.688,Z 557.067,A -85,B 0,C 180,E1 -7289.151,E2 -7289.151} C_VEL
LIN {X 0,Y 473.67,Z 557.281,A -85,B 0,C 180,E1 -7290.001,E2 -7290.001} C_VEL
LIN {X 0,Y 473.688,Z 557.063,A -85,B 0,C 180,E1 -7290.851,E2 -7290.851} C_VEL
LIN {X 0,Y 473.741,Z 555.459,A -85,B 0,C 180,E1 -7292.552,E2 -7292.552} C_VEL
LIN {X 0,Y 473.796,Z 554.059,A -85,B 0,C 180,E1 -7293.402,E2 -7293.402} C_VEL
LIN {X 0,Y 473.762,Z 551.114,A -85,B 0,C 180,E1 -7294.681,E2 -7294.681} C_VEL
LIN {X 0,Y 473.836,Z 547.128,A -85,B 0,C 180,E1 -7295.96,E2 -7295.96} C_VEL
LIN {X 0,Y 474.016,Z 540.994,A -85,B 0,C 180,E1 -7297.455,E2 -7297.455} C_VEL
LIN {X 0,Y 474.274,Z 534.293,A -85,B 0,C 180,E1 -7298.737,E2 -7298.737} C_VEL
LIN {X 0,Y 474.596,Z 525.967,A -85,B 0,C 180,E1 -7300.021,E2 -7300.021} C_VEL
LIN {X 0,Y 474.986,Z 517.414,A -85,B 0,C 180,E1 -7301.091,E2 -7301.091} C_VEL
LIN {X 0,Y 475.487,Z 507.062,A -85,B 0,C 180,E1 -7302.14,E2 -7302.14} C_VEL
LIN {X 0,Y 475.924,Z 495.082,A -85,B 0,C 180,E1 -7303.113,E2 -7303.113} C_VEL
LIN {X 0,Y 476.442,Z 482.88,A -85,B 0,C 180,E1 -7303.87,E2 -7303.87} C_VEL
LIN {X 0,Y 476.871,Z 470.318,A -85,B 0,C 180,E1 -7304.456,E2 -7304.456} C_VEL
LIN {X 0,Y 477.234,Z 458.201,A -85,B 0,C 180,E1 -7304.853,E2 -7304.853} C_VEL
LIN {X 0,Y 477.447,Z 444.72,A -85,B 0,C 180,E1 -7305.119,E2 -7305.119} C_VEL
LIN {X 0,Y 477.934,Z 361.757,A -85,B 0,C 180,E1 -7306.374,E2 -7306.374} C_VEL
LIN {X 0,Y 475.328,Z 344.791,A -85,B 0,C 180,E1 -7306.724,E2 -7306.724} C_VEL
LIN {X 0,Y 475.893,Z 328.15,A -85,B 0,C 180,E1 -7309.61,E2 -7309.61} C_VEL
LIN {X 0,Y 476.553,Z 311.388,A -85,B 0,C 180,E1 -7312.547,E2 -7312.547} C_VEL
LIN {X 0,Y 476.552,Z 306.245,A -85,B 0,C 180,E1 -7313.465,E2 -7313.465} C_VEL
LIN {X 0,Y 474.641,Z 296.365,A -85,B 0,C 180,E1 -7315.376,E2 -7315.376} C_VEL
LIN {X 0,Y 474.645,Z 296.359,A -85,B 0,C 180,E1 -7318.283,E2 -7318.283} C_VEL
LIN {X 0,Y 474.602,Z 296.362,A -85,B 0,C 180,E1 -7321.218,E2 -7321.218} C_VEL
LIN {X 0,Y 474.636,Z 296.362,A -85,B 0,C 180,E1 -7324.241,E2 -7324.241} C_VEL
